FUNCTION_BLOCK "SimaHydTO_AxisAdvanced_SyncAxis"   // FB33112, FBD
TITLE = SimaHydTO_AxisAdvanced_SyncAxis
{ S7_Optimized_Access := 'TRUE' }
FAMILY : SimaHydTO/LAxisBasics
VERSION : 1.0
// Function block information: See Function block network 1
// stored: AutoNumber true, IsIECCheckEnabled false, IsRetainMemResEnabled false, MemoryReserve 100, SetENOAutomatically false, UDAEnableTagReadback false
   VAR_INPUT
      axis : TO_SynchronousAxis;   // Technology object (axis)
      moveRelativeExecute : Bool;   // MC_MoveRelative: Start job with a positive edge
      moveRelativeDistance : LReal := 0.0;   // Distance of relative movement
      moveAbsoluteExecute : Bool;   // MC_MoveAbsolute: Start job with a positive edge
      moveAbsolutePosition : LReal := 0.0;   // Target position of absolute movement
      moveAbsoluteDirection : Int := 1;   // Direction of absolute movement: 0: Positive direction / 1: Negative direction / 3: Shortest direction
      moveAbsPositionControlled : Bool := true;   // 0: Non position-controlled operation / 1: Position-controlled mode - The parameter applies as long as the MC_MoveJog command is executed. After this, the setting of MC_Power applies again.
      haltExecute : Bool;   // MC_Halt: Start job with a positive edge
      haltAbortAcceleration : Bool := false;   // Acceleration control: False: The current acceleration at the start of the job is reduced using the configured jerk. Afterwards, the deceleration builds up / True: The acceleration is set to 0.0 at the start of the job, and the deceleration immediately builds up.
      Velocity : LReal := 100.0;   // Velocity of movement
      Acceleration : LReal := -1.0;   // Acceleration of movement
      Deceleration : LReal := -1.0;   // Deceleration of movement
      Jerk : LReal := -1.0;   // Jerk of movement
   END_VAR
   VAR_OUTPUT
      moveRelativeDone { ExternalWritable := 'False'} : Bool;   // MC_MoveRelative: Job is completed
      moveRelativeBusy { ExternalWritable := 'False'} : Bool;   // MC_MoveRelative: Job is running
      moveAbsoluteDone { ExternalWritable := 'False'} : Bool;   // MC_MoveAbsolute: Job is completed
      moveAbsoluteBusy { ExternalWritable := 'False'} : Bool;   // MC_MoveAbsolute: Job is running
      haltDone { ExternalWritable := 'False'} : Bool;   // MC_Halt: Job is running
      haltBusy { ExternalWritable := 'False'} : Bool;   // MC_Halt: Job is running
      commandAborted { ExternalWritable := 'False'} : Bool;   // The job was aborted by another job during execution (see also StatusID)
      error { ExternalWritable := 'False'} : Bool;   // An error occurred during execution of the job. The job is rejected. The cause of the error can be found in the "ErrorID" parameter.
      errorID { ExternalWritable := 'False'} : Word;   // ErrorID of motion control instruction (see also StatusID)
      statusID { ExternalWritable := 'False'} : Int;   // Additional specification of affected Motion control instruction of CommandAborted or Error: 0: No instruction / 1: MC_Power / 2: MC_Reset / 3: MC_Home / 4: MC_MoveJog
   END_VAR
   VAR
      instMcMoveRelative { ExternalAccessible := 'False'; ExternalVisible := 'False'; ExternalWritable := 'False'; S7_SetPoint := 'True'} : MC_MOVERELATIVE;   // PLCopen functions of basic motion control
      instMcMoveAbsolute { ExternalAccessible := 'False'; ExternalVisible := 'False'; ExternalWritable := 'False'; S7_SetPoint := 'True'} : MC_MOVEABSOLUTE;
      instMcHalt { ExternalAccessible := 'False'; ExternalVisible := 'False'; ExternalWritable := 'False'; S7_SetPoint := 'True'} : MC_HALT;
      statCommandAborted { ExternalAccessible := 'False'; ExternalVisible := 'False'; ExternalWritable := 'False'} : Array[#ARRAY_BEGIN..#ARRAY_END] of Bool;   // Arrays to save error information of PLCopen functions
      statError { ExternalAccessible := 'False'; ExternalVisible := 'False'; ExternalWritable := 'False'} : Array[#ARRAY_BEGIN..#ARRAY_END] of Bool;
      statErrorID { ExternalAccessible := 'False'; ExternalVisible := 'False'; ExternalWritable := 'False'} : Array[#ARRAY_BEGIN..#ARRAY_END] of Word;
      instMoveAbsOpenLoop { ExternalAccessible := 'False'; ExternalVisible := 'False'; ExternalWritable := 'False'; S7_SetPoint := 'True'} : "LSimaHydTO_MC_MoveAbsOpenLoop";
   END_VAR
   VAR_TEMP
      tempDwordCommandAborted : DWord;   // Variables to check error informations of PLCopen functions
      tempDwordError : DWord;
      tempCount : Int;   // Counter of FOR counting loop
   END_VAR
   VAR CONSTANT
      ARRAY_BEGIN : Int := 1;   // Start-Index of array (Maximum 32 Array elements!)
      ARRAY_END : Int := 32;   // End-Index of array (Maximum 32 Array elements!)
      ERROR_DEFAULT : Bool := false;   // Default values of output signals
      ERRORID_DEFAULT : Word := 16#0;
      STATUSID_DEFAULT : Int := 0;
   END_VAR
BEGIN

REGION Network 1 (SCL): Axis Basics - Header
   //=============================================================================
   //SIEMENS AG
   //(c)Copyright 2016 All Rights Reserved
   //-----------------------------------------------------------------------------
   //Library:       AxisAdvanced
   //Tested with:   S7-1500 V2.5
   //Engineering:   TIA Portal V15
   //Restrictions:  Motion Control Library V4.0
   //Requirements:  S7-1500(T)
   //Functionality: Advanced axis control of TO_SynchronousAxis
   //-----------------------------------------------------------------------------
   //Change log table:
   //Version  Date       Expert in charge Changes applied
   //01.00.00 19.07.2019 ArSc             First released version
   //=============================================================================
END_REGION

REGION Network 2: Axis Advanced - MC_MoveRelative
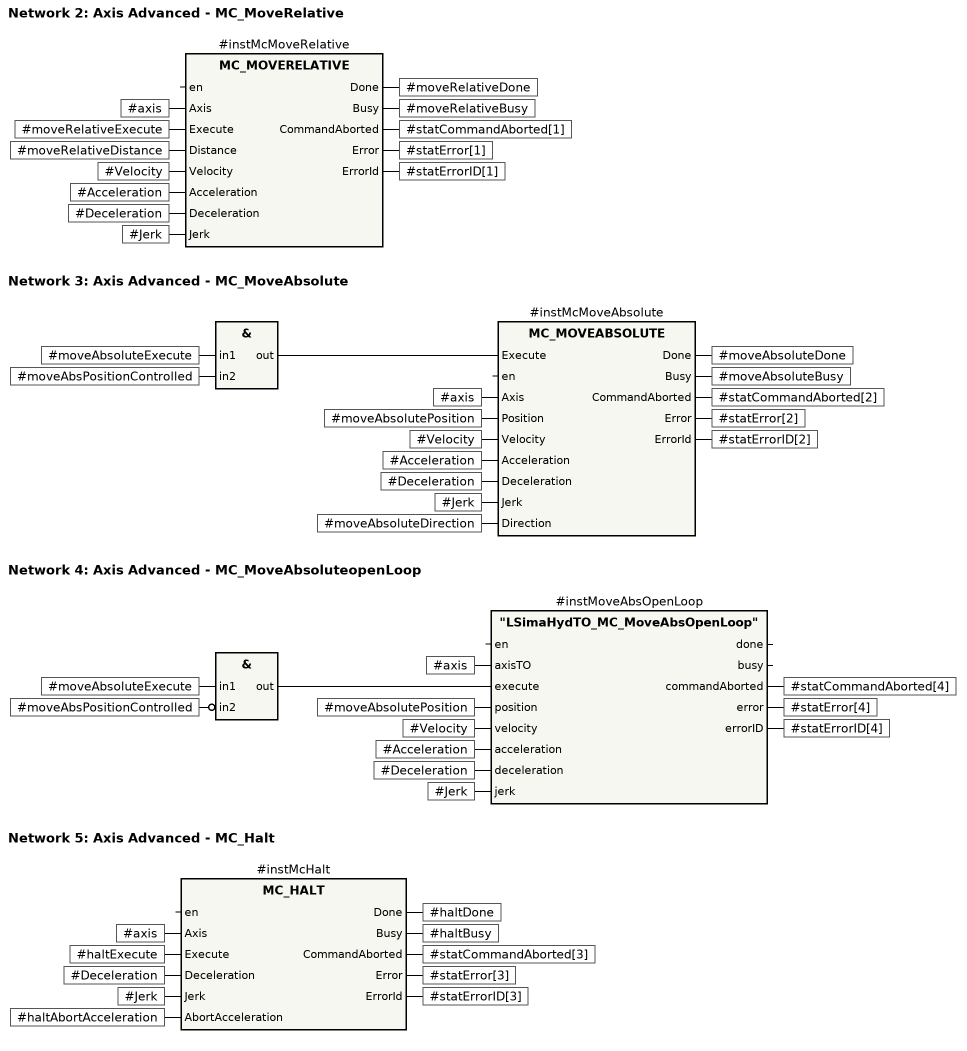
   #instMcMoveRelative(Axis := #axis,   // MC_MOVERELATIVE
                       Execute := #moveRelativeExecute,
                       Distance := #moveRelativeDistance,
                       Velocity := #Velocity,
                       Acceleration := #Acceleration,
                       Deceleration := #Deceleration,
                       Jerk := #Jerk,
                       Done => #moveRelativeDone,
                       Busy => #moveRelativeBusy,
                       CommandAborted => #statCommandAborted[1],
                       Error => #statError[1],
                       ErrorId => #statErrorID[1]);
END_REGION

REGION Network 3: Axis Advanced - MC_MoveAbsolute
   #instMcMoveAbsolute(Execute := #moveAbsoluteExecute AND #moveAbsPositionControlled,   // MC_MOVEABSOLUTE
                       Axis := #axis,
                       Position := #moveAbsolutePosition,
                       Velocity := #Velocity,
                       Acceleration := #Acceleration,
                       Deceleration := #Deceleration,
                       Jerk := #Jerk,
                       Direction := #moveAbsoluteDirection,
                       Done => #moveAbsoluteDone,
                       Busy => #moveAbsoluteBusy,
                       CommandAborted => #statCommandAborted[2],
                       Error => #statError[2],
                       ErrorId => #statErrorID[2]);
END_REGION

REGION Network 4: Axis Advanced - MC_MoveAbsoluteopenLoop
   #instMoveAbsOpenLoop(axisTO := #axis,   // "LSimaHydTO_MC_MoveAbsOpenLoop"
                        execute := #moveAbsoluteExecute AND NOT #moveAbsPositionControlled,
                        position := #moveAbsolutePosition,
                        velocity := #Velocity,
                        acceleration := #Acceleration,
                        deceleration := #Deceleration,
                        jerk := #Jerk,
                        commandAborted => #statCommandAborted[4],
                        error => #statError[4],
                        errorID => #statErrorID[4]);
END_REGION

REGION Network 5: Axis Advanced - MC_Halt
   #instMcHalt(Axis := #axis,   // MC_HALT
               Execute := #haltExecute,
               Deceleration := #Deceleration,
               Jerk := #Jerk,
               AbortAcceleration := #haltAbortAcceleration,
               Done => #haltDone,
               Busy => #haltBusy,
               CommandAborted => #statCommandAborted[3],
               Error => #statError[3],
               ErrorId => #statErrorID[3]);
END_REGION

REGION Network 6 (SCL): Axis Basics - Generate output signals and error detection
   //General output signals

   //Reset output signals
   #commandAborted := False;
   #error := False;
   #errorID := #ERRORID_DEFAULT;
   #statusID := #STATUSID_DEFAULT;

   //Transfer ARRAY to DWORD
   GATHER(IN:=#statCommandAborted,
          OUT=>#tempDwordCommandAborted);
   GATHER(IN:=#statError,
          OUT=>#tempDwordError);

   //Check for errors or command aborts
   IF (#tempDwordError > DWORD#0)
   THEN
     //Select error information
     FOR #tempCount := #ARRAY_BEGIN TO #ARRAY_END
     DO
       IF (#statError[#tempCount] = True)
       THEN
         #error := True;
         #errorID := #statErrorID[#tempCount];
         #statusID := #tempCount;
         EXIT;
       END_IF;
     END_FOR;
   ELSIF (#tempDwordCommandAborted > DWORD#0)
   THEN
     //Select command aborted information
     FOR #tempCount := #ARRAY_BEGIN TO #ARRAY_END
     DO
       IF (#statCommandAborted[#tempCount] = True)
       THEN
         #commandAborted := True;
         #errorID := #statErrorID[#tempCount];
         #statusID := #tempCount;
         EXIT;
       END_IF;
     END_FOR;
   END_IF;
END_REGION
END_FUNCTION_BLOCK

FUNCTION_BLOCK "SimaHydTO_ParameterSettings"
{ S7_Optimized_Access := 'TRUE' }
FAMILY : SimaHydTO
VERSION : 1.0
   VAR_IN_OUT 
      hmiConnection : "SimaHydTO_typeHMIConnection";
      axisData : "LSimaHydTO_typeAxisData";
      VCharArray : Array[*] of "SimaHydTO_typeVCharArray";
   END_VAR

   VAR 
      statSaveDBL { ExternalAccessible := 'False'; ExternalVisible := 'False'; ExternalWritable := 'False'} : Bool;
      statLoadDBL { ExternalAccessible := 'False'; ExternalVisible := 'False'; ExternalWritable := 'False'} : Bool;
      statEditOld { ExternalAccessible := 'False'; ExternalVisible := 'False'; ExternalWritable := 'False'} : Bool;
      statActivateOld { ExternalAccessible := 'False'; ExternalVisible := 'False'; ExternalWritable := 'False'} : Bool;
      statAbortOld { ExternalAccessible := 'False'; ExternalVisible := 'False'; ExternalWritable := 'False'} : Bool;
      statRestoreOld { ExternalAccessible := 'False'; ExternalVisible := 'False'; ExternalWritable := 'False'} : Bool;
      statApplayOld { ExternalAccessible := 'False'; ExternalVisible := 'False'; ExternalWritable := 'False'} : Bool;
      statDefaultAxisData { ExternalAccessible := 'False'; ExternalVisible := 'False'; ExternalWritable := 'False'} : "SimaHydTO_typeHMIConnectionParameterSettingsAxisData";
      instMC_WriteToROM { ExternalAccessible := 'False'; ExternalVisible := 'False'; ExternalWritable := 'False'} : "LSimaHydTO_MC_WriteToROM";
      instMC_ReadFromROM { ExternalAccessible := 'False'; ExternalVisible := 'False'; ExternalWritable := 'False'} : "LSimaHydTO_MC_ReadFromROM";
      instVCharSelector { ExternalAccessible := 'False'; ExternalVisible := 'False'; ExternalWritable := 'False'} : "SimaHydTO_HmiVCharSelector";
      statSaveOld { ExternalAccessible := 'False'; ExternalVisible := 'False'; ExternalWritable := 'False'} : Bool;
   END_VAR

   VAR_TEMP 
      tempVariant : Variant;
      tempErrorVariant : Int;
      tempDbAny : DB_ANY;
      tempVCharData : REF_TO "LSimaHydTO_typeVCharData";
   END_VAR


BEGIN
	//=============================================================================
	//SIEMENS AG
	//(c)Copyright 2016 All Rights Reserved
	//-----------------------------------------------------------------------------
	//Library:       SimaHydTO_ParameterSettings
	//Tested with:   S7-1500 V2.5
	//Engineering:   TIA Portal V15
	//Restrictions:  -
	//Requirements:  S7-1500(T)
	//Functionality: Manipulate parameter data of selected hydraulic axis
	//-----------------------------------------------------------------------------
	//Change log table:
	//Version  Date       Expert in charge Changes applied
	//01.00.00 17.07.2019 ArSc             First released version
	//=============================================================================
	
	
	IF (#hmiConnection.AxisSelector.Status.selectionChanged
	    OR #instMC_ReadFromROM.done)
	    OR (#hmiConnection.ParameterSettings.Commands.Edit
	    AND NOT #statEditOld
	    AND NOT #hmiConnection.ParameterSettings.Status.EditorActive)
	THEN
	    IF #hmiConnection.AxisSelector.Status.dataValid THEN
	        //Convert data
	        //Get data from axis
	        #hmiConnection.ParameterSettings.AxisData.Actor := #axisData.Actor;
	        #hmiConnection.ParameterSettings.AxisData.ValveCharacteristic := #axisData.ValveCharacteristic;
	        #hmiConnection.ParameterSettings.AxisData.ForceLimits := #axisData.ForceLimits;
	        #hmiConnection.ParameterSettings.AxisData.Pressure_A_Transducer := #axisData.Pressure_A_Transducer;
	        #hmiConnection.ParameterSettings.AxisData.Pressure_B_Transducer := #axisData.Pressure_B_Transducer;
	        #hmiConnection.ParameterSettings.AxisData.PositionControl := #axisData.PositionControl;
	        #hmiConnection.ParameterSettings.AxisData.ForceControl := #axisData.ForceControl;
	        #hmiConnection.ParameterSettings.AxisData.DynamicAxisModel := #axisData.DynamicAxisModel;
	        #hmiConnection.ParameterSettings.AxisData.SmoothingFilter := #axisData.SmoothingFilter;
	        #hmiConnection.ParameterSettings.AxisData.Name := #axisData.Name;
	        IF #axisData.ValveCharacteristic.DB_NUMBER > 0 THEN
	            #tempDbAny := #axisData.ValveCharacteristic.DB_NUMBER;
	            #tempVariant := DB_ANY_TO_VARIANT(in := #tempDbAny, err => #tempErrorVariant);
	            
	            IF TypeOf(#tempVariant) = LSimaHydTO_typeVCharData THEN
	                #tempVCharData ?= #tempVariant;
	                #hmiConnection.ParameterSettings.AxisData.VCharName := #tempVCharData^.Name;
	            ELSE
	                #hmiConnection.ParameterSettings.AxisData.VCharName := wstring#'';
	            END_IF;
	        ELSE
	            #hmiConnection.ParameterSettings.AxisData.VCharName := wstring#'';
	        END_IF;
	        
	    ELSE
	        #hmiConnection.ParameterSettings.AxisData := #statDefaultAxisData;
	    END_IF;
	    IF #hmiConnection.AxisSelector.Status.selectionChanged THEN
	        #hmiConnection.ParameterSettings.Status.EditorActive := False;
	    END_IF;
	    
	END_IF;
	
	//Open parameter data
	IF (#hmiConnection.ParameterSettings.Commands.Edit
	    AND NOT #statEditOld
	    AND NOT #hmiConnection.ParameterSettings.Status.EditorActive
	    AND #hmiConnection.AxisSelector.Status.dataValid)
	THEN
	    #hmiConnection.ParameterSettings.Status.EditorActive := True;
	END_IF;
	
	//Save parameter data
	IF ((#hmiConnection.ParameterSettings.Commands.Activate AND NOT #statActivateOld)
	    OR (#hmiConnection.ParameterSettings.Commands.Save AND NOT #statSaveOld))
	    AND #hmiConnection.ParameterSettings.Status.EditorActive
	    AND #hmiConnection.AxisSelector.Status.dataValid
	THEN
	    //Write back axis data
	    #hmiConnection.ParameterSettings.Status.StateActivation := 1;
	    
	    #axisData.Actor := #hmiConnection.ParameterSettings.AxisData.Actor;
	    #axisData.ValveCharacteristic := #hmiConnection.ParameterSettings.AxisData.ValveCharacteristic;
	    #axisData.ForceLimits := #hmiConnection.ParameterSettings.AxisData.ForceLimits;
	    #axisData.Pressure_A_Transducer := #hmiConnection.ParameterSettings.AxisData.Pressure_A_Transducer;
	    #axisData.Pressure_B_Transducer := #hmiConnection.ParameterSettings.AxisData.Pressure_B_Transducer;
	    #axisData.PositionControl := #hmiConnection.ParameterSettings.AxisData.PositionControl;
	    #axisData.ForceControl := #hmiConnection.ParameterSettings.AxisData.ForceControl;
	    #axisData.DynamicAxisModel := #hmiConnection.ParameterSettings.AxisData.DynamicAxisModel;
	    #axisData.SmoothingFilter := #hmiConnection.ParameterSettings.AxisData.SmoothingFilter;
	    #axisData.Name := #hmiConnection.ParameterSettings.AxisData.Name;
	    //  save to load memory
	    #hmiConnection.ParameterSettings.Status.EditorActive := False;
	    #hmiConnection.ParameterSettings.Status.StateActivation := 0;
	    #hmiConnection.ParameterSettings.Status.StateLoading := 0;
	END_IF;
	
	IF #hmiConnection.ParameterSettings.Commands.Save
	    //AND #hmiConnection.ParameterSettings.Status.StateActivation = 1
	    AND #hmiConnection.AxisSelector.Status.dataValid
	    AND NOT #statSaveOld
	THEN
	    #statSaveDBL := TRUE;
	    
	END_IF;
	
	#instMC_WriteToROM(execute := #statSaveDBL,
	                   axis := #axisData);
	
	IF #instMC_WriteToROM.busy THEN
	    #hmiConnection.ParameterSettings.Status.StateSaving := 1;
	ELSIF #instMC_WriteToROM.error THEN
	    #hmiConnection.ParameterSettings.Status.StateSaving := 2;
	    #statSaveDBL := FALSE;
	    
	ELSE
	    #hmiConnection.ParameterSettings.Status.StateSaving := 0;
	    #statSaveDBL := FALSE;
	    
	END_IF;
	
	
	IF (#hmiConnection.ParameterSettings.Commands.Restore
	    AND NOT #statRestoreOld)
	    AND #hmiConnection.AxisSelector.Status.dataValid
	THEN
	    #hmiConnection.ParameterSettings.Status.StateActivation := 0;
	    #hmiConnection.ParameterSettings.Status.StateSaving := 0;
	    #hmiConnection.ParameterSettings.Status.StateLoading := 1;
	    
	    #statLoadDBL := true;
	END_IF;
	#instMC_ReadFromROM(execute := #statLoadDBL,
	                    axis := #axisData);
	
	IF NOT #instMC_ReadFromROM.busy THEN
	    IF #instMC_ReadFromROM.done THEN
	        #hmiConnection.ParameterSettings.Status.StateActivation := 0;
	        #hmiConnection.ParameterSettings.Status.StateLoading := 0;
	    ELSIF #instMC_ReadFromROM.error THEN
	        #hmiConnection.ParameterSettings.Status.StateLoading := 2;
	    END_IF;
	    
	    
	    #statLoadDBL := FALSE;
	END_IF;
	
	
	//Abort parameter data
	IF (#hmiConnection.ParameterSettings.Commands.Abort
	    AND #hmiConnection.ParameterSettings.Status.EditorActive)
	THEN
	    //Reset output singal
	    #hmiConnection.ParameterSettings.Status.EditorActive := False;
	END_IF;
	
	
	//Save data from last cycle
	#statAbortOld := #hmiConnection.ParameterSettings.Commands.Abort;
	#statActivateOld := #hmiConnection.ParameterSettings.Commands.Activate;
	#statEditOld := #hmiConnection.ParameterSettings.Commands.Edit;
	#statRestoreOld := #hmiConnection.ParameterSettings.Commands.Restore;
	#statSaveOld := #hmiConnection.ParameterSettings.Commands.Save;
	
END_FUNCTION_BLOCK

FUNCTION_BLOCK "LSimaHydTO_MC_WriteToROM"
{ S7_Optimized_Access := 'TRUE' }
AUTHOR : APC_ERLF
FAMILY : LSimaHydTO
VERSION : 1.0
   VAR_INPUT 
      execute : Bool;
      parameter : Int;
   END_VAR

   VAR_OUTPUT 
      busy { ExternalWritable := 'False'} : Bool;
      done { ExternalWritable := 'False'} : Bool;
      commandAborted { ExternalWritable := 'False'} : Bool;
      error { ExternalWritable := 'False'} : Bool;
      errorID { ExternalWritable := 'False'} : Int;
   END_VAR

   VAR_IN_OUT 
      axis : "LSimaHydTO_typeAxisData";
   END_VAR

   VAR 
      statState { ExternalAccessible := 'False'; ExternalVisible := 'False'; ExternalWritable := 'False'} : DInt;
      statExecuteOld { ExternalAccessible := 'False'; ExternalVisible := 'False'; ExternalWritable := 'False'} : Bool;
      statBusyWrit { ExternalAccessible := 'False'; ExternalVisible := 'False'; ExternalWritable := 'False'} : Bool;
      statBusy { ExternalAccessible := 'False'; ExternalVisible := 'False'; ExternalWritable := 'False'} : Bool;
      statRetVal { ExternalAccessible := 'False'; ExternalVisible := 'False'; ExternalWritable := 'False'} : Int;
   END_VAR

   VAR_TEMP 
      tempVarParameter : Variant;
   END_VAR

   VAR CONSTANT 
      STATE_IDLE : DInt := 0;
      LAST_PARAM : DInt := 10;
   END_VAR


BEGIN
	//================================================================================
	//SIEMENS AG // (c)Copyright 2019 All Rights Reserved
	//--------------------------------------------------------------------------------
	//Library:       LSimaHydTO
	//Tested with:   S7-15xx
	//Engineering:   TIA Portal  V15
	//Restrictions:  -
	//Requirements:  S7-1500 (FW 2.5)
	//Functionality: Write parameter from RAM into ROM 
	//
	//--------------------------------------------------------------------------------
	//Change log table:
	//
	//Version     Date          Expert in charge    Changes applied
	//01.00.00    15.03.2018    APC_ERLF            First released version
	//================================================================================
	
	
	IF #execute AND NOT #statExecuteOld THEN
	  #done := FALSE;
	  #statBusy := TRUE;
	  #statBusyWrit := FALSE;
	  #error := FALSE;
	  #errorID := 0;
	  IF #parameter = 0 OR #parameter = 1 THEN
	    #statState := 1;
	  ELSE
	    #statState := #parameter;
	  END_IF;
	END_IF;
	IF #statBusy THEN
	  
	  CASE #statState OF
	      
	    1: // actor
	      
	      #statRetVal := WRIT_DBL(REQ := TRUE, SRCBLK := #axis.Actor, BUSY => #statBusyWrit, DSTBLK => #axis.Actor);
	      
	      
	    2: // valve characteristic
	      
	      #statRetVal := WRIT_DBL(REQ := TRUE, SRCBLK := #axis.ValveCharacteristic, BUSY => #statBusyWrit, DSTBLK => #axis.ValveCharacteristic);
	      
	      
	    3: // force limits
	      
	      #statRetVal := WRIT_DBL(REQ := TRUE, SRCBLK := #axis.ForceLimits, BUSY => #statBusyWrit, DSTBLK => #axis.ForceLimits);
	      
	      
	    4: // A-transducer
	      
	      #statRetVal := WRIT_DBL(REQ := TRUE, SRCBLK := #axis.Pressure_A_Transducer, BUSY => #statBusyWrit, DSTBLK => #axis.Pressure_A_Transducer);
	      
	      
	    5: // B-transducer
	      
	      #statRetVal := WRIT_DBL(REQ := TRUE, SRCBLK := #axis.Pressure_B_Transducer, BUSY => #statBusyWrit, DSTBLK => #axis.Pressure_B_Transducer);
	      
	      
	    6: // position control
	      
	      #statRetVal := WRIT_DBL(REQ := TRUE, SRCBLK := #axis.PositionControl, BUSY => #statBusyWrit, DSTBLK => #axis.PositionControl);
	      
	      
	    7: // force control
	      
	      #statRetVal := WRIT_DBL(REQ := TRUE, SRCBLK := #axis.ForceControl, BUSY => #statBusyWrit, DSTBLK => #axis.ForceControl);
	      
	      
	    8: // dynamic axis model
	      
	      #statRetVal := WRIT_DBL(REQ := TRUE, SRCBLK := #axis.DynamicAxisModel, BUSY => #statBusyWrit, DSTBLK => #axis.DynamicAxisModel);
	      
	      
	    9: // smoothing filter
	      
	      #statRetVal := WRIT_DBL(REQ := TRUE, SRCBLK := #axis.SmoothingFilter, BUSY => #statBusyWrit, DSTBLK => #axis.SmoothingFilter);
	      
	      
	    10: // name
	      
	      #statRetVal := WRIT_DBL(REQ := TRUE, SRCBLK := #axis.Name, BUSY => #statBusyWrit, DSTBLK => #axis.Name);
	      
	      
	    ELSE
	      #statState := #STATE_IDLE;
	      #statBusy := FALSE;
	  END_CASE;
	  
	  IF NOT #statBusyWrit THEN
	    IF #statRetVal = 0 THEN
	      IF #parameter = 0 AND #statState < #LAST_PARAM THEN
	        #statState := 1 + #statState;
	      ELSE
	        #statBusy := false;
	        #done := TRUE;
	      END_IF;
	    ELSE
	      #statBusy := FALSE;
	      #error := TRUE;
	      #errorID := #statRetVal;
	      #statState := #STATE_IDLE;
	    END_IF;
	  END_IF;
	ELSIF NOT #execute THEN
	  #done := FALSE;
	  #error := FALSE;
	  #errorID := 0;
	END_IF;
	#statExecuteOld := #execute;
	#busy := #statBusy;
	
END_FUNCTION_BLOCK

FUNCTION_BLOCK "LSimaHydTO_MC_ReadFromROM"
{ S7_Optimized_Access := 'TRUE' }
AUTHOR : APC_ERLF
FAMILY : LSimaHydTO
VERSION : 1.0
   VAR_INPUT 
      execute : Bool;
      parameter : Int;
   END_VAR

   VAR_OUTPUT 
      busy { ExternalWritable := 'False'} : Bool;
      done { ExternalWritable := 'False'} : Bool;
      commandAborted { ExternalWritable := 'False'} : Bool;
      error { ExternalWritable := 'False'} : Bool;
      errorID { ExternalWritable := 'False'} : Word;
   END_VAR

   VAR_IN_OUT 
      axis : "LSimaHydTO_typeAxisData";
   END_VAR

   VAR 
      statState { ExternalAccessible := 'False'; ExternalVisible := 'False'; ExternalWritable := 'False'} : DInt;
      statExecuteOld { ExternalAccessible := 'False'; ExternalVisible := 'False'; ExternalWritable := 'False'} : Bool;
      statBusyRead { ExternalAccessible := 'False'; ExternalVisible := 'False'; ExternalWritable := 'False'} : Bool;
      statRetVal { ExternalAccessible := 'False'; ExternalVisible := 'False'; ExternalWritable := 'False'} : Int;
   END_VAR

   VAR_TEMP 
      tempVarParameter : Variant;
   END_VAR

   VAR CONSTANT 
      STATE_IDLE : DInt := 0;
      LAST_PARAM : DInt := 10;
   END_VAR


BEGIN
	//================================================================================
	//SIEMENS AG // (c)Copyright 2019 All Rights Reserved
	//--------------------------------------------------------------------------------
	//Library:       LSimaHydTO
	//Tested with:   S7-15xx
	//Engineering:   TIA Portal  V15
	//Restrictions:  -
	//Requirements:  S7-1500 (FW 2.5)
	//Functionality: Read parameter from ROM into RAM 
	//
	//--------------------------------------------------------------------------------
	//Change log table:
	//
	//Version     Date          Expert in charge    Changes applied
	//01.00.00    15.03.2018    APC_ERLF            First released version
	//================================================================================
	
	
	IF #execute AND NOT #statExecuteOld THEN
	  #done := FALSE;
	  #busy := TRUE;
	  #statBusyRead := TRUE;
	  #error := FALSE;
	  #errorID := 0;
	  IF #parameter = 0 OR #parameter = 1 THEN
	    #statState := 1;
	  ELSE
	    #statState := #parameter;
	  END_IF;
	END_IF;
	IF #statBusyRead THEN
	  
	  CASE #statState OF
	      
	    1: // actor
	      
	      #statRetVal := READ_DBL(REQ := TRUE, SRCBLK := #axis.Actor, BUSY => #statBusyRead, DSTBLK => #axis.Actor);
	      
	      
	    2: // valve characteristic
	      
	      #statRetVal := READ_DBL(REQ := TRUE, SRCBLK := #axis.ValveCharacteristic, BUSY => #statBusyRead, DSTBLK => #axis.ValveCharacteristic);
	      
	      
	    3: // force limits
	      
	      #statRetVal := READ_DBL(REQ := TRUE, SRCBLK := #axis.ForceLimits, BUSY => #statBusyRead, DSTBLK => #axis.ForceLimits);
	      
	      
	    4: // ring transducer
	      
	      #statRetVal := READ_DBL(REQ := TRUE, SRCBLK := #axis.Pressure_A_Transducer, BUSY => #statBusyRead, DSTBLK => #axis.Pressure_A_Transducer);
	      
	      
	    5: // piston transducer
	      
	      #statRetVal := READ_DBL(REQ := TRUE, SRCBLK := #axis.Pressure_B_Transducer, BUSY => #statBusyRead, DSTBLK => #axis.Pressure_B_Transducer);
	      
	      
	    6: // position control
	      
	      #statRetVal := READ_DBL(REQ := TRUE, SRCBLK := #axis.PositionControl, BUSY => #statBusyRead, DSTBLK => #axis.PositionControl);
	      
	      
	    7: // force control
	      
	      #statRetVal := READ_DBL(REQ := TRUE, SRCBLK := #axis.ForceControl, BUSY => #statBusyRead, DSTBLK => #axis.ForceControl);
	      
	      
	    8: // dynamic axis model
	      
	      #statRetVal := READ_DBL(REQ := TRUE, SRCBLK := #axis.DynamicAxisModel, BUSY => #statBusyRead, DSTBLK => #axis.DynamicAxisModel);
	      
	      
	    9: // smoothing filter
	      
	      #statRetVal := READ_DBL(REQ := TRUE, SRCBLK := #axis.SmoothingFilter, BUSY => #statBusyRead, DSTBLK => #axis.SmoothingFilter);
	      
	      
	    10: // name
	      
	      #statRetVal := READ_DBL(REQ := TRUE, SRCBLK := #axis.Name, BUSY => #statBusyRead, DSTBLK => #axis.Name);
	      
	      
	    ELSE
	      #statState := #STATE_IDLE;
	      #statBusyRead := FALSE;
	  END_CASE;
	  
	  IF NOT #statBusyRead THEN
	    IF #statRetVal = 0 THEN
	      IF #parameter = 0 AND #statState < #LAST_PARAM THEN
	        #statState := 1 + #statState;
	        #statBusyRead := TRUE;
	      ELSE
	        #busy := false;
	        #done := TRUE;
	      END_IF;
	    ELSE
	      #busy := FALSE;
	      #error := TRUE;
	      #errorID := INT_TO_WORD(#statRetVal);
	      #statState := #STATE_IDLE;
	    END_IF;
	  END_IF;
	ELSIF NOT #execute THEN
	  #done := FALSE;
	  #error := FALSE;
	  #errorID := 0;
	END_IF;
	#statExecuteOld := #execute;
	
END_FUNCTION_BLOCK

FUNCTION_BLOCK "SimaHydTO_FindObjects"
{ S7_Optimized_Access := 'TRUE' }
FAMILY : SimaHydTO
VERSION : 1.0
   VAR_INPUT 
      execute : Bool;
   END_VAR

   VAR_OUTPUT 
      done { ExternalWritable := 'False'} : Bool;
      busy { ExternalWritable := 'False'} : Bool;
      error { ExternalWritable := 'False'} : Bool;
      status { ExternalWritable := 'False'} : Word := #STATUS_NO_CALL;
   END_VAR

   VAR_IN_OUT 
      axesArray : Array[*] of "SimaHydTO_typeAxesArray";
      vCharArray : Array[*] of "SimaHydTO_typeVCharArray";
   END_VAR

   VAR 
      statAxesArrMinIndex { ExternalAccessible := 'False'; ExternalVisible := 'False'; ExternalWritable := 'False'} : Int;
      statAxesArrMaxIndex { ExternalAccessible := 'False'; ExternalVisible := 'False'; ExternalWritable := 'False'} : Int;
      statVCharArrMinIndex { ExternalAccessible := 'False'; ExternalVisible := 'False'; ExternalWritable := 'False'} : Int;
      statVCharArrMaxIndex { ExternalAccessible := 'False'; ExternalVisible := 'False'; ExternalWritable := 'False'} : Int;
      statVCharArrayFull { ExternalAccessible := 'False'; ExternalVisible := 'False'; ExternalWritable := 'False'} : Bool;
      statAxesArrayFull { ExternalAccessible := 'False'; ExternalVisible := 'False'; ExternalWritable := 'False'} : Bool;
      statExecuteOld { ExternalAccessible := 'False'; ExternalVisible := 'False'; ExternalWritable := 'False'} : Bool;
      statDone { ExternalAccessible := 'False'; ExternalVisible := 'False'; ExternalWritable := 'False'} : Bool;
      statBusy { ExternalAccessible := 'False'; ExternalVisible := 'False'; ExternalWritable := 'False'} : Bool;
      statError { ExternalAccessible := 'False'; ExternalVisible := 'False'; ExternalWritable := 'False'} : Bool;
      statStatus { ExternalAccessible := 'False'; ExternalVisible := 'False'; ExternalWritable := 'False'} : Word := #STATUS_NO_CALL;
      statFBState { ExternalAccessible := 'False'; ExternalVisible := 'False'; ExternalWritable := 'False'} : DInt := #FB_STATE_NO_PROCESSING;
      statActDB_NUMBER { ExternalAccessible := 'False'; ExternalVisible := 'False'; ExternalWritable := 'False'} : UInt;
      statRunTime { ExternalAccessible := 'False'; ExternalVisible := 'False'; ExternalWritable := 'False'} : LReal;
      statMemStart { ExternalAccessible := 'False'; ExternalVisible := 'False'; ExternalWritable := 'False'} : LReal;
      statMem { ExternalAccessible := 'False'; ExternalVisible := 'False'; ExternalWritable := 'False'} : LReal;
   END_VAR

   VAR_TEMP 
      tempExecute : Bool;
      tempInt : Int;
      tempInitDone : Bool;
   END_VAR

   VAR CONSTANT 
      FB_STATE_NO_PROCESSING : DInt := 0;
      FB_STATE_PROCESSING : DInt := 2;
      STATUS_EXECUTION_FINISHED : Word := 16#0000;
      STATUS_NO_CALL : Word := 16#7000;
      STATUS_FIRST_CALL : Word := 16#7001;
      STATUS_SUBSEQUENT_CALL : Word := 16#7002;
      ERR_UNDEFINED_STATE : Word := 16#8600;
   END_VAR


BEGIN
	//=============================================================================
	//SIEMENS AG
	//(c)Copyright 2016 All Rights Reserved
	//-----------------------------------------------------------------------------
	//Library:       SimaHydTO_HMI
	//Tested with:   S7-1500 V2.5
	//Engineering:   TIA Portal V15
	//Restrictions:  -
	//Requirements:  S7-1500(T)
	//Functionality: Search for hydraulic axes and valve charachteristics in project
	//-----------------------------------------------------------------------------
	//Change log table:
	//Version  Date       Expert in charge Changes applied
	//01.00.00 12.07.2019 ArSc             First released version
	//=============================================================================
	
	#tempExecute := #execute; // Work with temporary value / create process image
	
	REGION TRIGGERING
	    IF (#tempExecute = TRUE) AND (#statExecuteOld = FALSE) // Check if FB is triggered
	        
	    THEN // First call; initialize FB
	        #statDone := FALSE;
	        #statBusy := TRUE;
	        #statError := FALSE;
	        #statStatus := #STATUS_FIRST_CALL;
	        
	        #statAxesArrMinIndex := DINT_TO_INT(LOWER_BOUND(ARR := #axesArray, DIM := 1));
	        #statAxesArrMaxIndex := DINT_TO_INT(UPPER_BOUND(ARR := #axesArray, DIM := 1));
	        #statVCharArrMinIndex := DINT_TO_INT(LOWER_BOUND(ARR := #vCharArray, DIM := 1));
	        #statVCharArrMaxIndex := DINT_TO_INT(UPPER_BOUND(ARR := #vCharArray, DIM := 1));
	        
	        #statVCharArrayFull := FALSE;
	        #statAxesArrayFull := FALSE;
	        #statActDB_NUMBER := 1;
	        
	        #statFBState := #FB_STATE_PROCESSING; // State machine - start processing
	        
	    ELSIF (#statStatus = #STATUS_FIRST_CALL) THEN
	        #statStatus := #STATUS_SUBSEQUENT_CALL;
	    END_IF;
	    
	    // Edge detection 'execute' input
	    #statExecuteOld := #tempExecute;
	END_REGION TRIGGERING
	
	IF (#statStatus = #STATUS_NO_CALL) THEN // Nothing to do -> End here to reduce "system load"
	    RETURN;
	END_IF;
	
	REGION STATE_MACHINE
	    CASE #statFBState OF // State machine of FB
	        #FB_STATE_NO_PROCESSING: // No processing active (Note: this state must always be present and left empty)
	            ;
	            
	        #FB_STATE_PROCESSING:
	            // Processing active
	            // 
	            #statRunTime := RUNTIME(MEM := #statMemStart);
	            
	            REPEAT
	                IF TypeOfDB(#statActDB_NUMBER) = LSimaHydTO_typeVCharData THEN
	                    // enter vchar to data exchange
	                    #tempInitDone := FALSE;
	                    FOR #tempInt := #statVCharArrMinIndex TO #statVCharArrMaxIndex DO
	                        IF #vCharArray[#tempInt].VChar_DB = #statActDB_NUMBER THEN
	                            #vCharArray[#tempInt].initialized := TRUE;
	                            #tempInitDone := TRUE;
	                            EXIT;
	                        END_IF;
	                    END_FOR;
	                    IF NOT #tempInitDone THEN
	                        FOR #tempInt := #statVCharArrMinIndex TO #statVCharArrMaxIndex DO
	                            IF NOT #vCharArray[#tempInt].initialized THEN
	                                #vCharArray[#tempInt].VChar_DB := #statActDB_NUMBER;
	                                #vCharArray[#tempInt].initialized := TRUE;
	                                #tempInitDone := TRUE;
	                                EXIT;
	                            END_IF;
	                            IF #tempInt = #statVCharArrMaxIndex THEN
	                                #statVCharArrayFull := TRUE;
	                            END_IF;
	                            
	                        END_FOR;
	                    END_IF;
	                    
	                ELSIF TypeOfDB(#statActDB_NUMBER) = LSimaHydTO_typeAxisData THEN
	                    #tempInitDone := FALSE;
	                    FOR #tempInt := #statAxesArrMinIndex TO #statAxesArrMaxIndex DO
	                        IF #axesArray[#tempInt].axisData = #statActDB_NUMBER THEN
	                            #axesArray[#tempInt].initialized := TRUE;
	                            #tempInitDone := TRUE;
	                            EXIT;
	                        END_IF;
	                    END_FOR;
	                    IF NOT #tempInitDone THEN
	                        FOR #tempInt := #statAxesArrMinIndex TO #statAxesArrMaxIndex DO
	                            IF NOT #axesArray[#tempInt].initialized THEN
	                                #axesArray[#tempInt].axisData := #statActDB_NUMBER;
	                                #axesArray[#tempInt].initialized := TRUE;
	                                #tempInitDone := TRUE;
	                                EXIT;
	                            END_IF;
	                            IF #tempInt = #statAxesArrMaxIndex THEN
	                                #statAxesArrayFull := TRUE;
	                            END_IF;
	                        END_FOR;
	                    END_IF;
	                    
	                END_IF;
	                IF #statAxesArrayFull AND #statVCharArrayFull THEN
	                    #statBusy := FALSE;
	                    #statStatus := #STATUS_EXECUTION_FINISHED;
	                END_IF;
	                
	                IF #statStatus = #STATUS_SUBSEQUENT_CALL THEN
	                    IF #statActDB_NUMBER < uint#65_535 THEN
	                        #statActDB_NUMBER += 1;
	                    ELSE
	                        #statBusy := FALSE;
	                        #statStatus := #STATUS_EXECUTION_FINISHED;
	                    END_IF;
	                END_IF;
	                #statMem := #statMemStart;
	                #statRunTime := RUNTIME(MEM := #statMem);
	            UNTIL NOT #statBusy OR #statRunTime > 0.01 // interupt after 10 ms
	            END_REPEAT;
	            
	            
	        ELSE // Undefined state in state machine reached
	            #statStatus := #ERR_UNDEFINED_STATE;
	    END_CASE;
	END_REGION STATE_MACHINE
	
	REGION OUTPUTS
	    // Write outputs
	    IF (#statStatus = #STATUS_EXECUTION_FINISHED) AND (#statDone = FALSE) THEN // Execution finished without errors
	        #statDone := TRUE;
	        #statBusy := FALSE;
	        #statError := FALSE;
	        #statFBState := #FB_STATE_NO_PROCESSING; // Switch state machine to "no processing"
	        
	    ELSIF (#statStatus.%X15 = TRUE) AND (#statError = FALSE) THEN // Error occurred (#statStatus is 16#8000 to 16#FFFF)
	        #statDone := FALSE;
	        #statBusy := FALSE;
	        #statError := TRUE;
	        #statFBState := #FB_STATE_NO_PROCESSING; // Switch state machine to "no processing"
	        
	    ELSIF (#tempExecute = FALSE) AND ((#statDone = TRUE) OR (#statError = TRUE)) THEN // Reset outputs
	        #statDone := FALSE;
	        #statBusy := FALSE;
	        #statError := FALSE;
	        #statStatus := #STATUS_NO_CALL;
	    END_IF;
	    
	    // Write static values to outputs
	    #done := #statDone;
	    #busy := #statBusy;
	    #error := #statError;
	    #status := #statStatus;
	END_REGION OUTPUTS
END_FUNCTION_BLOCK

FUNCTION_BLOCK "SimaHydTO_VCharManagement"
{ S7_Optimized_Access := 'TRUE' }
FAMILY : SimaHydTO
VERSION : 1.0
   VAR_IN_OUT 
      hmiConnection : "SimaHydTO_typeHMIConnection";
      axisData : "LSimaHydTO_typeAxisData";
      vCharArray : Array[*] of "SimaHydTO_typeVCharArray";
   END_VAR

   VAR 
      statSaveDBL { ExternalAccessible := 'False'; ExternalVisible := 'False'; ExternalWritable := 'False'} : Bool;
      statLoadDBL { ExternalAccessible := 'False'; ExternalVisible := 'False'; ExternalWritable := 'False'} : Bool;
      statEditOld { ExternalAccessible := 'False'; ExternalVisible := 'False'; ExternalWritable := 'False'} : Bool;
      statActivateOld { ExternalAccessible := 'False'; ExternalVisible := 'False'; ExternalWritable := 'False'} : Bool;
      statAbortOld { ExternalAccessible := 'False'; ExternalVisible := 'False'; ExternalWritable := 'False'} : Bool;
      statRestoreOld { ExternalAccessible := 'False'; ExternalVisible := 'False'; ExternalWritable := 'False'} : Bool;
      statApplayOld { ExternalAccessible := 'False'; ExternalVisible := 'False'; ExternalWritable := 'False'} : Bool;
      statDefaultAxisData { ExternalAccessible := 'False'; ExternalVisible := 'False'; ExternalWritable := 'False'} : "SimaHydTO_typeHMIConnectionParameterSettingsAxisData";
      instMC_WriteToROM { ExternalAccessible := 'False'; ExternalVisible := 'False'; ExternalWritable := 'False'} : "LSimaHydTO_MC_WriteToROM";
      instMC_ReadFromROM { ExternalAccessible := 'False'; ExternalVisible := 'False'; ExternalWritable := 'False'} : "LSimaHydTO_MC_ReadFromROM";
      instVCharSelector { ExternalAccessible := 'False'; ExternalVisible := 'False'; ExternalWritable := 'False'} : "SimaHydTO_HmiVCharSelector";
      statSaveOld { ExternalAccessible := 'False'; ExternalVisible := 'False'; ExternalWritable := 'False'} : Bool;
   END_VAR

   VAR_TEMP 
      tempVariant : Variant;
      tempErrorVariant : Int;
      tempDbAny : DB_ANY;
      tempVCharData : REF_TO "LSimaHydTO_typeVCharData";
   END_VAR


BEGIN
	//=============================================================================
	//SIEMENS AG
	//(c)Copyright 2016 All Rights Reserved
	//-----------------------------------------------------------------------------
	//Library:       SimaHydTO_VCharManagement
	//Tested with:   S7-1500 V2.5
	//Engineering:   TIA Portal V15
	//Restrictions:  -
	//Requirements:  S7-1500(T)
	//Functionality: Manipulate active VChar of selected hydraulic axis
	//-----------------------------------------------------------------------------
	//Change log table:
	//Version  Date       Expert in charge Changes applied
	//01.00.00 17.07.2019 ArSc             First released version
	//=============================================================================
	
	  // Vchar selection
	  #instVCharSelector(command:=#hmiConnection.ParameterSettings.Commands.VCharSelector,
	                       status:=#hmiConnection.ParameterSettings.Status.VCharSelector,
	                       vCharArray:=#vCharArray);
	  
	  
	  IF #hmiConnection.ParameterSettings.Commands.ApplyVChar
	    AND NOT #statApplayOld
	    AND #hmiConnection.ParameterSettings.Status.VCharSelector.dataValid
	  THEN
	    #axisData.ValveCharacteristic.DB_NUMBER := #hmiConnection.ParameterSettings.Status.VCharSelector.selectedVChar;
	    #hmiConnection.AxisSelector.Status.selectedVChar := #hmiConnection.ParameterSettings.Status.VCharSelector.selectedVChar;
	    #hmiConnection.AxisSelector.Status.selectedVCharInteger := DB_ANY_TO_UINT(#hmiConnection.ParameterSettings.Status.VCharSelector.selectedVChar);
	    
	    
	    #hmiConnection.ParameterSettings.AxisData.VCharName := #hmiConnection.ParameterSettings.Status.VCharSelector.selectedVCharName;
	    #hmiConnection.ParameterSettings.AxisData.ValveCharacteristic.DB_NUMBER := #hmiConnection.ParameterSettings.Status.VCharSelector.selectedVChar;
	    
	    #hmiConnection.AxisSelector.Status.selectedVCharName := #hmiConnection.ParameterSettings.Status.VCharSelector.selectedVCharName;
	    
	    
	    
	  END_IF;
	
	#statApplayOld := #hmiConnection.ParameterSettings.Commands.ApplyVChar;
	
END_FUNCTION_BLOCK

FUNCTION "SimaHydTO_GetAxisToUnits_PosAxis" : "SimaHydTO_typeHMIConnectionAxisToDataAxisUnits"
{ S7_Optimized_Access := 'TRUE' }
FAMILY : SimaHydTO
VERSION : 1.0
   VAR_INPUT 
      axisTO {InstructionName := 'TO_PositioningAxis'; LibVersion := '4.0'} : TO_PositioningAxis;
   END_VAR


BEGIN
	//=============================================================================
	//SIEMENS AG
	//(c)Copyright 2016 All Rights Reserved
	//-----------------------------------------------------------------------------
	//Library:       SimaHyd_AxisBasics
	//Tested with:   S7-1500 V2.5
	//Engineering:   TIA Portal V15
	//Restrictions:  Motion Control Library V4.0
	//Requirements:  S7-1500(T)
	//Functionality: Get axis units of TO_PositioningAxis
	//-----------------------------------------------------------------------------
	//Change log table:
	//Version  Date       Expert in charge Changes applied
	//01.00.00 20.05.2019 ArSc             First released version
	//=============================================================================
	
	
	//-----------------------------------------------------------------------------
	//Write axis units
	//-----------------------------------------------------------------------------
	
	#SimaHydTO_GetAxisToUnits_PosAxis.forceUnit := #axisTO.Units.ForceUnit;
	#SimaHydTO_GetAxisToUnits_PosAxis.lengthUnit := #axisTO.Units.LengthUnit;
	#SimaHydTO_GetAxisToUnits_PosAxis.velocityUnit := #axisTO.Units.VelocityUnit;
	
END_FUNCTION

FUNCTION "SimaHydTO_GetAxisToUnits_SyncAxis" : "SimaHydTO_typeHMIConnectionAxisToDataAxisUnits"
{ S7_Optimized_Access := 'TRUE' }
FAMILY : SimaHydTO
VERSION : 1.0
   VAR_INPUT 
      axisTO {InstructionName := 'TO_SynchronousAxis'; LibVersion := '4.0'} : TO_SynchronousAxis;
   END_VAR


BEGIN
	//=============================================================================
	//SIEMENS AG
	//(c)Copyright 2016 All Rights Reserved
	//-----------------------------------------------------------------------------
	//Library:       SimaHyd_AxisBasics
	//Tested with:   S7-1500 V2.5
	//Engineering:   TIA Portal V15
	//Restrictions:  Motion Control Library V4.0
	//Requirements:  S7-1500(T)
	//Functionality: Get axis units of TO_SynchronousAxis
	//-----------------------------------------------------------------------------
	//Change log table:
	//Version  Date       Expert in charge Changes applied
	//01.00.00 20.05.2019 ArSc             First released version
	//=============================================================================
	
	
	//-----------------------------------------------------------------------------
	//Write axis data
	//-----------------------------------------------------------------------------
	#SimaHydTO_GetAxisToUnits_SyncAxis := "SimaHydTO_GetAxisToUnits_PosAxis"(#axisTO);
END_FUNCTION

FUNCTION "SimaHydTO_HmiAxisAnimation" : Void
{ S7_Optimized_Access := 'TRUE' }
FAMILY : SimaHydTO
VERSION : 1.0
   VAR_IN_OUT 
      hmiConnection : "SimaHydTO_typeHMIConnection";
      axisData : "LSimaHydTO_typeAxisData";
   END_VAR

   VAR_TEMP 
      tempPositionLimitsSW : "LSimaHydTO_typePositionLimits";
      tempTravelDistance : LReal;
   END_VAR


BEGIN
	//=============================================================================
	//SIEMENS AG
	//(c)Copyright 2016 All Rights Reserved
	//-----------------------------------------------------------------------------
	//Library:       SimaHydTO_HMI
	//Tested with:   S7-1500 V2.5
	//Engineering:   TIA Portal V15
	//Restrictions:  -
	//Requirements:  S7-1500(T)
	//Functionality: Transfer data from/to HMI to/from selected axis
	//-----------------------------------------------------------------------------
	//Change log table:
	//Version  Date       Expert in charge Changes applied
	//01.00.00 12.07.2019 ArSc             First released version
	//=============================================================================
	
	
	// 
	IF #hmiConnection.AxisSelector.Status.dataValid 
	THEN
	  //Read data
	  //Check data
	  IF #axisData.DataInitialized = TRUE
	  THEN
	    //Calculate HMI data
	    #tempPositionLimitsSW := #axisData.Internal.PositionLimits_SW;
	    IF (#tempPositionLimitsSW.Active = True)
	    THEN
	      #hmiConnection.HmiData.MinPosition := #tempPositionLimitsSW.MinPosition;
	      #hmiConnection.HmiData.MaxPosition := #tempPositionLimitsSW.MaxPosition;
	      #tempTravelDistance := (#tempPositionLimitsSW.MaxPosition - #tempPositionLimitsSW.MinPosition);
	      //Calculate percent value
	      IF (#tempTravelDistance > 0.0)
	      THEN
	        #hmiConnection.HmiData.ActualPositionPercent := DINT_TO_INT(TRUNC(100.0 * ((#axisData.ActualPosition - #tempPositionLimitsSW.MinPosition) /
	                                                            #tempTravelDistance)));
	        
	        #hmiConnection.HmiData.SafetyDistanceAnimation := #tempPositionLimitsSW.MinPosition + #hmiConnection.BasicAxisControl.ControlDirectOutput.safetyDistance;
	
	    
	
	      ELSE
	          #hmiConnection.HmiData.ActualPositionPercent := 0;
	          #hmiConnection.HmiData.SafetyDistanceAnimation := 0.0;
	      END_IF;
	    ELSE
	      #hmiConnection.HmiData.MinPosition := 0.0;
	      #hmiConnection.HmiData.MaxPosition := 0.0;
	      #hmiConnection.HmiData.ActualPositionPercent := 0;
	      #hmiConnection.HmiData.SafetyDistanceAnimation := 0.0;
	      #hmiConnection.HmiData.selectedAxis := 0;
	      #hmiConnection.HmiData.selectedAxisTO := 0;
	    END_IF;
	  END_IF;
	  #hmiConnection.AxisData.Force := #axisData.Force;
	  #hmiConnection.AxisData.Velocity := #axisData.Velocity;
	  #hmiConnection.AxisData.Position := #axisData.Position;
	  #hmiConnection.AxisData.ActualForce := #axisData.ActualForce;
	  #hmiConnection.AxisData.ActualVelocity := #axisData.ActualVelocity;
	  #hmiConnection.AxisData.ActualPosition := #axisData.ActualPosition;
	  #hmiConnection.AxisData.Status_A_Transducer.PressureValue := #axisData.Status_A_Transducer.PressureValue;
	  #hmiConnection.AxisData.Status_B_Transducer.PressureValue := #axisData.Status_B_Transducer.PressureValue;
	  #hmiConnection.AxisData.StatusActor := #axisData.StatusActor;
	  
	END_IF;
	
END_FUNCTION

FUNCTION "LSimaHydTO_AreaToDiameter" : Void
{ S7_Optimized_Access := 'TRUE' }
AUTHOR : APC_ERLF
FAMILY : LSimaHydTO
VERSION : 1.0
   VAR_INPUT 
      pistonArea : LReal;
      pistonRodArea : LReal;
   END_VAR

   VAR_OUTPUT 
      pistonDiameter : LReal;
      pistonRodDiameter : LReal;
   END_VAR


BEGIN
	//================================================================================
	//SIEMENS AG // (c)Copyright 2019 All Rights Reserved
	//--------------------------------------------------------------------------------
	//Library:       LSimaHydTO
	//Tested with:   S7-15xx
	//Engineering:   TIA Portal  V15
	//Restrictions:  -
	//Requirements:  S7-1500 (FW 2.5)
	//Functionality: HMI support program - Internal use  
	//
	//--------------------------------------------------------------------------------
	//Change log table:
	//
	//Version     Date          Expert in charge    Changes applied
	//01.00.00    15.03.2018    APC_ERLF            First released version
	//================================================================================
	
	
	IF #pistonArea > 0.0 THEN
	  #pistonDiameter := SQRT(#pistonArea * 1.2732395);
	  IF #pistonRodArea > 0.0 AND #pistonRodArea < #pistonArea THEN
	    #pistonRodDiameter := SQRT(#pistonDiameter*#pistonDiameter -  #pistonRodArea * 1.2732395);
	  ELSE
	    #pistonRodDiameter := 0.0;
	  END_IF;
	ELSE
	  #pistonRodDiameter := 0.0;
	  #pistonDiameter := 0.0;
	END_IF;
	
	
END_FUNCTION

FUNCTION "LSimaHydTO_Covariance" : Int
{ S7_Optimized_Access := 'TRUE' }
AUTHOR : APC_ERLF
FAMILY : LSimaHydTO
VERSION : 1.0
   VAR_INPUT 
      firstIdx : Int;
      numOfPoints : Int;
   END_VAR

   VAR_OUTPUT 
      factor : Real;
      correlation : Real;
   END_VAR

   VAR_IN_OUT 
      valuesX : Array[*] of Real;
      valuesY : Array[*] of Real;
   END_VAR

   VAR_TEMP 
      i : Int;
      ret : Int;
      sum2X : Real;
      sum2Y : Real;
      meanValueX : Real;
      meanValueY : Real;
      sumX : Real;
      sumY : Real;
      varianceX : Real;
      variancey : Real;
      sumCoVar : Real;
      covariance : Real;
      tempLB : Int;
      tempUB : Int;
      lastIdx : Int;
   END_VAR


BEGIN
	//================================================================================
	//SIEMENS AG // (c)Copyright 2019 All Rights Reserved
	//--------------------------------------------------------------------------------
	//Library:       LSimaHydTO
	//Tested with:   S7-15xx
	//Engineering:   TIA Portal  V15
	//Restrictions:  -
	//Requirements:  S7-1500 (FW 2.5)
	//Functionality: HMI support program - Internal use  
	//
	//--------------------------------------------------------------------------------
	//Change log table:
	//
	//Version     Date          Expert in charge    Changes applied
	//01.00.00    15.03.2018    APC_ERLF            First released version
	//================================================================================
	
	
	IF #numOfPoints < 2 THEN
	  #LSimaHydTO_Covariance := -1;
	  RETURN;
	END_IF;
	#tempLB := DINT_TO_INT(MAX(IN1 := LOWER_BOUND(ARR:=#valuesX, DIM:=1),IN2 := LOWER_BOUND(ARR:=#valuesY, DIM:=1)));
	#tempUB := DINT_TO_INT(MIN(IN1 := UPPER_BOUND(ARR := #valuesX, DIM := 1), IN2 := UPPER_BOUND(ARR := #valuesY, DIM := 1)));
	#lastIdx := #firstIdx + #numOfPoints - 1;
	IF #tempLB > #firstIdx  THEN
	  #ret := -2;
	ELSIF #tempUB < #lastIdx THEN
	  #ret := -3;
	ELSE
	  #ret := 0;
	  #sumX := 0.0;
	  #sumY := 0.0;
	  #sum2X := 0.0;
	  #sum2Y := 0.0;
	  #sumCoVar := 0.0;
	  FOR #i := #firstIdx TO #lastIdx DO
	    #sumX := #sumX + #valuesX[#i];
	    #sumY := #sumY + #valuesY[#i];
	  END_FOR;
	  #meanValueX := #sumX / #numOfPoints;
	  #meanValueY := #sumY / #numOfPoints;
	  FOR #i := #firstIdx TO #lastIdx DO
	    #sum2X := #sum2X + SQR(#valuesX[#i] - #meanValueX);
	    #sum2Y := #sum2Y + SQR(#valuesY[#i] - #meanValueY);
	    #sumCoVar := #sumCoVar + (#valuesX[#i] - #meanValueX) * (#valuesY[#i] - #meanValueY);
	  END_FOR;
	  #varianceX := #sum2X / (#numOfPoints - 1);
	  #variancey := #sum2Y / (#numOfPoints - 1);
	  #covariance := #sumCoVar / (#numOfPoints - 1);
	  #factor := #covariance / #varianceX;
	  #correlation := #covariance / (SQRT(#varianceX) * SQRT(#variancey));
	END_IF;
	#LSimaHydTO_Covariance := #ret;
	
	
END_FUNCTION

FUNCTION "LSimaHydTO_DiameterToArea" : Void
{ S7_Optimized_Access := 'TRUE' }
AUTHOR : APC_ERLF
FAMILY : LSimaHydTO
VERSION : 1.0
   VAR_INPUT 
      pistonDiameter : LReal;
      pistonRodDiameter : LReal;
   END_VAR

   VAR_OUTPUT 
      pistonArea : LReal;
      pistonRodArea : LReal;
   END_VAR


BEGIN
	//================================================================================
	//SIEMENS AG // (c)Copyright 2019 All Rights Reserved
	//--------------------------------------------------------------------------------
	//Library:       LSimaHydTO
	//Tested with:   S7-15xx
	//Engineering:   TIA Portal  V15
	//Restrictions:  -
	//Requirements:  S7-1500 (FW 2.5)
	//Functionality: HMI support program - Internal use  
	//
	//--------------------------------------------------------------------------------
	//Change log table:
	//
	//Version     Date          Expert in charge    Changes applied
	//01.00.00    15.03.2018    APC_ERLF            First released version
	//================================================================================
	
	
	IF #pistonDiameter > 0.0 THEN
	  #pistonArea := #pistonDiameter*#pistonDiameter * 0.7853981;
	  IF #pistonRodDiameter > 0.0 AND #pistonRodDiameter < #pistonDiameter THEN
	    #pistonRodArea := (#pistonDiameter*#pistonDiameter -  #pistonRodDiameter*#pistonRodDiameter) * 0.7853981;
	  ELSE
	    #pistonRodArea := 0.0;
	  END_IF;
	ELSE
	  #pistonRodArea := 0.0;
	  #pistonArea := 0.0;
	END_IF;
	
	
END_FUNCTION

FUNCTION "LSimaHydTO_GetAxisForceCommandState" : Word
{ S7_Optimized_Access := 'TRUE' }
AUTHOR : APC_ERLF
FAMILY : LSimaHydTO
VERSION : 1.0
   VAR_INPUT 
      commandID : UDInt;
   END_VAR

   VAR_IN_OUT 
      axis : "LSimaHydTO_typeAxisData";
   END_VAR

   VAR_TEMP 
      tempRetVal : Word;
   END_VAR

   VAR CONSTANT 
      MOTION_STATE_NOT_EXISTEND : Word := 16#0000;
      MOTION_STATE_BUFFERED_OR_MOTION : Word := 16#0001;
      MOTION_STATE_EXECUTED : Word := 16#0010;
      MOTION_STATE_ABORTED : Word := 16#0020;
      MOTION_STATE_ERROR : Word := 16#8000;
   END_VAR


BEGIN
	//================================================================================
	//SIEMENS AG // (c)Copyright 2019 All Rights Reserved
	//--------------------------------------------------------------------------------
	//Library:       LSimaHydTO
	//Tested with:   S7-15xx
	//Engineering:   TIA Portal  V15
	//Restrictions:  -
	//Requirements:  S7-1500 (FW 2.5)
	//Functionality: - for internal use
	//
	//--------------------------------------------------------------------------------
	//Change log table:
	//
	//Version     Date          Expert in charge    Changes applied
	//01.00.00    15.03.2018    APC_ERLF            First released version
	//================================================================================
	
	
	IF #axis.Internal.Control.ForceCommand.commandID = #commandID THEN
	  #tempRetVal := #MOTION_STATE_BUFFERED_OR_MOTION;
	ELSIF #axis.Internal.MotionData.ForceCmdTracking.CommandID = #commandID THEN
	  IF (#axis.Internal.MotionData.ForceCmdTracking.State AND #MOTION_STATE_BUFFERED_OR_MOTION) <> 0 THEN
	    #tempRetVal := #MOTION_STATE_BUFFERED_OR_MOTION;
	  ELSE
	    #tempRetVal := #axis.Internal.MotionData.ForceCmdTracking.State;
	  END_IF;
	ELSE
	  #tempRetVal := #MOTION_STATE_NOT_EXISTEND;
	END_IF;
	#LSimaHydTO_GetAxisForceCommandState := #tempRetVal;
	
	
END_FUNCTION

FUNCTION "LSimaHydTO_GetCommandID" : UDInt
{ S7_Optimized_Access := 'TRUE' }
AUTHOR : APC_ERLF
FAMILY : LSimaHydTO
VERSION : 1.0
   VAR_IN_OUT 
      axis : "LSimaHydTO_typeAxisData";
   END_VAR


BEGIN
	//================================================================================
	//SIEMENS AG // (c)Copyright 2019 All Rights Reserved
	//--------------------------------------------------------------------------------
	//Library:       LSimaHydTO
	//Tested with:   S7-15xx
	//Engineering:   TIA Portal  V15
	//Restrictions:  -
	//Requirements:  S7-1500 (FW 2.5)
	//Functionality: - for internal use
	//
	//--------------------------------------------------------------------------------
	//Change log table:
	//
	//Version     Date          Expert in charge    Changes applied
	//01.00.00    15.03.2018    APC_ERLF            First released version
	//================================================================================
	
	
	#axis.Internal.CommandIDPool := #axis.Internal.CommandIDPool+1;
	IF #axis.Internal.CommandIDPool = 0 THEN
	  #axis.Internal.CommandIDPool := #axis.Internal.CommandIDPool + 1;
	END_IF;
	#LSimaHydTO_GetCommandID:= #axis.Internal.CommandIDPool;
	
	
END_FUNCTION

FUNCTION "LSimaHydTO_GetPosAxisData" : Void
{ S7_Optimized_Access := 'TRUE' }
AUTHOR : APC_ERLF
FAMILY : LSimaHydTO
VERSION : 1.0
   VAR_INPUT 
      axisTO {InstructionName := 'TO_PositioningAxis'; LibVersion := '4.0'} : TO_PositioningAxis;
   END_VAR

   VAR_OUTPUT 
      statusWord : DWord;
      errorWord : DWord;
      errorDetail : "LSimaHydTO_typeErrorDetail";
      velocity : LReal;
      acceleration : LReal;
      position : LReal;
      actualSpeed : LReal;
      actualVelocity : LReal;
      actualAcceleration : LReal;
      actualPosition : LReal;
      referenceSpeed : LReal;
      positionLimits_SW {InstructionName := 'TO_Struct_PositionLimitsSW'; LibVersion := '4.0'} : TO_Struct_PositionLimitsSW;
      dynamicLimits : "LSimaHydTO_typeDynamicLimits";
   END_VAR


BEGIN
	//================================================================================
	//SIEMENS AG // (c)Copyright 2019 All Rights Reserved
	//--------------------------------------------------------------------------------
	//Library:       LSimaHydTO
	//Tested with:   S7-15xx
	//Engineering:   TIA Portal  V15
	//Restrictions:  -
	//Requirements:  S7-1500 (FW 2.5)
	//Functionality: - for internal use
	//
	//--------------------------------------------------------------------------------
	//Change log table:
	//
	//Version     Date          Expert in charge    Changes applied
	//01.00.00    15.03.2018    APC_ERLF            First released version
	//================================================================================
	
	#statusWord := #axisTO.StatusWord;
	#errorWord := #axisTO.ErrorWord;
	#velocity := #axisTO.Velocity;
	#acceleration := #axisTO.Acceleration;
	#position := #axisTO.Position;
	#actualSpeed := #axisTO.ActualSpeed;
	#actualVelocity := #axisTO.ActualVelocity;
	#actualAcceleration := #axisTO.#ActualAcceleration;
	#actualPosition := #axisTO.ActualPosition;
	#referenceSpeed := #axisTO.Actor.DriveParameter.ReferenceSpeed;
	#errorDetail.Number := #axisTO.ErrorDetail.Number;
	#errorDetail.Reaction := #axisTO.ErrorDetail.Reaction;
	//software limit switches
	#positionLimits_SW.Active := #axisTO.PositionLimits_SW.Active;
	#positionLimits_SW.MaxPosition := #axisTO.PositionLimits_SW.MaxPosition;
	#positionLimits_SW.MinPosition := #axisTO.PositionLimits_SW.MinPosition;
	#dynamicLimits.MaxVelocity := MIN(IN1 := #axisTO.DynamicLimits.MaxVelocity, IN2 := #axisTO.DynamicLimits.Velocity);
	#dynamicLimits.MaxAcceleration := #axisTO.DynamicLimits.MaxAcceleration;
	#dynamicLimits.MaxDeceleration := #axisTO.DynamicLimits.MaxDeceleration;
	#dynamicLimits.MaxJerk := #axisTO.DynamicLimits.MaxJerk;
	
	
END_FUNCTION

FUNCTION_BLOCK "LSimaHydTO_HandleDBL"
{ S7_Optimized_Access := 'TRUE' }
AUTHOR : APC_ERLF
FAMILY : LSimaHydTO
VERSION : 1.0
   VAR_INPUT 
      executeRead : Bool;
      executeWrite : Bool;
   END_VAR

   VAR_OUTPUT 
      busy { ExternalWritable := 'False'} : Bool;
      done { ExternalWritable := 'False'} : Bool;
      error { ExternalWritable := 'False'} : Bool;
      errorID { ExternalWritable := 'False'} : Int;
   END_VAR

   VAR_IN_OUT 
      memoryDB : Variant;
      cardDB : Variant;
   END_VAR

   VAR 
      statFBState { ExternalAccessible := 'False'; ExternalVisible := 'False'; ExternalWritable := 'False'} : Int;
      statExecuteReadOld { ExternalAccessible := 'False'; ExternalVisible := 'False'; ExternalWritable := 'False'} : Bool;
      statExecuteWriteOld { ExternalAccessible := 'False'; ExternalVisible := 'False'; ExternalWritable := 'False'} : Bool;
      statRetVal { ExternalAccessible := 'False'; ExternalVisible := 'False'; ExternalWritable := 'False'} : Int;
   END_VAR

   VAR CONSTANT 
      FB_STATE_IDLE : Int;
      FB_STATE_READ : Int := 10;
      FB_STATE_WRITE : Int := 20;
      FB_STATE_ERROR : Int := 100;
   END_VAR


BEGIN
	//================================================================================
	//SIEMENS AG // (c)Copyright 2019 All Rights Reserved
	//--------------------------------------------------------------------------------
	//Library:       LSimaHydTO
	//Tested with:   S7-15xx
	//Engineering:   TIA Portal  V15 (SW 2.5)
	//Restrictions:  -
	//Requirements:  S7-1500
	//Functionality: Save and load DB data to/from card
	//
	//--------------------------------------------------------------------------------
	//Change log table:
	//
	//Version     Date          Expert in charge    Changes applied
	//01.00.00    15.03.2018    APC_ERLF            First released version
	//================================================================================
	
	
	CASE #statFBState OF
	    
	  #FB_STATE_IDLE: 
	
	    IF #executeRead AND NOT #statExecuteReadOld THEN
	      #busy := false;
	      #done := false;
	      #error := false;
	      #errorID := 0;
	      #statRetVal := READ_DBL(REQ := #executeRead, SRCBLK := #cardDB, BUSY => #busy, DSTBLK => #memoryDB);
	      IF #busy THEN
	        #statFBState := #FB_STATE_READ;
	      ELSE
	        #error := TRUE;
	        #errorID := #statRetVal;
	        #statFBState := #FB_STATE_ERROR;
	      END_IF;
	    ELSIF  #executeWrite AND NOT #statExecuteWriteOld THEN
	      #busy := false;
	      #done := false;
	      #error := false;
	      #errorID := 0;
	      #statRetVal := WRIT_DBL(REQ := #executeWrite, SRCBLK :=#memoryDB , BUSY => #busy, DSTBLK => #cardDB);
	      IF #busy THEN
	        #statFBState := #FB_STATE_WRITE;
	      ELSE
	        #error := TRUE;
	        #errorID := #statRetVal;
	        #statFBState := #FB_STATE_ERROR;
	      END_IF;
	    ELSIF NOT(#executeRead OR #executeWrite) THEN
	      #done := FALSE;
	      #busy := FALSE;
	    END_IF;
	    
	    
	  #FB_STATE_READ:
	    
	    #statRetVal := READ_DBL(REQ := #executeRead, SRCBLK := #cardDB, BUSY => #busy, DSTBLK => #memoryDB);;
	    IF NOT #busy THEN
	      IF #statRetVal = 0 THEN
	        #done := TRUE;
	        #statFBState := #FB_STATE_IDLE;
	      ELSE
	        #error := TRUE;
	        #errorID := #statRetVal;
	        #statFBState := #FB_STATE_ERROR;
	      END_IF;
	    END_IF;
	    
	    
	  #FB_STATE_WRITE:
	    
	    #statRetVal := WRIT_DBL(REQ := #executeWrite, SRCBLK :=#memoryDB , BUSY => #busy, DSTBLK => #cardDB);
	    IF NOT #busy THEN
	      IF #statRetVal = 0 THEN
	        #done := TRUE;
	        #statFBState := #FB_STATE_IDLE;
	      ELSE
	        #error := TRUE;
	        #errorID := #statRetVal;
	        #statFBState := #FB_STATE_ERROR;
	      END_IF;
	    END_IF;
	    
	    
	  #FB_STATE_ERROR:
	    
	    IF NOT (#executeRead OR #executeWrite) THEN
	      #statFBState := #FB_STATE_IDLE;
	    END_IF;
	  ELSE
	    ;
	END_CASE;
	
	#statExecuteReadOld := #executeRead;
	#statExecuteWriteOld := #executeWrite;
	
	
END_FUNCTION_BLOCK

FUNCTION_BLOCK "LSimaHydTO_MC_ForceControl"
{ S7_Optimized_Access := 'TRUE' }
AUTHOR : APC_ERLF
FAMILY : LSimaHydTO
VERSION : 1.0
   VAR_INPUT 
      execute : Bool;
      forceControlProfile : UInt;
      mode : DInt;
      forceProfileMode : DInt;
      conditionMode : DInt := 1;
      compareMode : DInt := 1;
      conditionValue : LReal;
      forceValue : LReal;
      forceDerivedValue : LReal;
      velocityLimitingValue : LReal;
   END_VAR

   VAR_OUTPUT 
      done { ExternalWritable := 'False'} : Bool;
      inForceControl { ExternalWritable := 'False'} : Bool;
      busy { ExternalWritable := 'False'} : Bool;
      commandAborted { ExternalWritable := 'False'} : Bool;
      error { ExternalWritable := 'False'} : Bool;
      errorID { ExternalWritable := 'False'} : Word;
   END_VAR

   VAR_IN_OUT 
      axis : "LSimaHydTO_typeAxisData";
   END_VAR

   VAR 
      statFBState { ExternalAccessible := 'False'; ExternalVisible := 'False'; ExternalWritable := 'False'} : DInt;
      statCommandID { ExternalAccessible := 'False'; ExternalVisible := 'False'; ExternalWritable := 'False'} : UDInt;
      statCmdState { ExternalAccessible := 'False'; ExternalVisible := 'False'; ExternalWritable := 'False'} : Word;
      statExecuteOld { ExternalAccessible := 'False'; ExternalVisible := 'False'; ExternalWritable := 'False'} : Bool;
   END_VAR

   VAR CONSTANT 
      NO_ERROR : Word := 16#0000;
      STATE_IDLE : DInt;
      STATE_FIRST_CYCLE : DInt := 10;
      STATE_BUSY : DInt := 20;
      STATE_DONE : DInt := 30;
      STATE_COMMAND_ABORTED : DInt := 40;
      STATE_ERROR : DInt := 100;
      MOTION_STATE_NOT_EXISTEND : Word := 16#0000;
      MOTION_STATE_BUFFERED_OR_MOTION : Word := 16#0001;
      MOTION_STATE_EXECUTED : Word := 16#0010;
      MOTION_STATE_ABORTED : Word := 16#0020;
      MOTION_STATE_ERROR : Word := 16#8000;
      NO_ERROR_REACTION : DInt := 0;
      ALARM_AXIS_ERROR_OCCURED : Word := 16#8001;
      ALARM_WRONG_MODE : Word := 16#800A;
      ALARM_AXIS_DISABLED : Word := 16#800F;
      ALARM_FORCE_PROFILE_MODE : Word := 16#80B1;
      ALARM_CONDITION_MODE : Word := 16#80B2;
      ALARM_FORCE_PROFILE : Word := 16#80B3;
      ALARM_COMPARE_MODE : Word := 16#80B4;
      ALARM_FORCE_DERIVED_VALUE : Word := 16#80B5;
   END_VAR


BEGIN
	//================================================================================
	//SIEMENS AG // (c)Copyright 2019 All Rights Reserved
	//--------------------------------------------------------------------------------
	//Library:       LSimaHydTO
	//Tested with:   S7-15xx
	//Engineering:   TIA Portal  V15
	//Restrictions:  -
	//Requirements:  S7-1500 (FW 2.5)
	//Functionality: Function to activate and deactivate pressure control mode for an axis.
	//               In addition, you can specify the conditions under which pressure
	//               control becomes active.
	//
	//--------------------------------------------------------------------------------
	//Change log table:
	//
	//Version     Date          Expert in charge    Changes applied
	//01.00.00    15.03.2018    APC_ERLF            First released version
	//================================================================================
	
	
	//----------------------------------------------------------------------
	//start
	//----------------------------------------------------------------------
	
	//rising edge of execute starts functionality
	IF #execute AND NOT #statExecuteOld THEN
	  //initialization
	  #done := FALSE;
	  #commandAborted := FALSE;
	  #inForceControl := FALSE;
	  #busy := FALSE;
	  #error := FALSE;
	  #errorID := #NO_ERROR;
	  #statFBState := #STATE_FIRST_CYCLE;
	END_IF;
	
	
	//----------------------------------------------------------------------
	//busy
	//----------------------------------------------------------------------
	
	CASE #statFBState OF
	    
	  #STATE_FIRST_CYCLE:
	    
	    //==================================================================
	    //This state runs just one time after a rising edge on execute and
	    //calls the function to start the motion.
	    //Get a commandId and buffer it for tracking the command in the
	    //following state STATE_BUSY
	    //==================================================================
	    
	    #commandAborted := FALSE;
	    IF #mode < 0 OR #mode > 2 THEN
	      #error := TRUE;
	      #errorID := #ALARM_WRONG_MODE;
	      #statFBState := #STATE_ERROR;
	    ELSIF #mode <> 0 AND (#forceProfileMode < 0 OR #forceProfileMode > 2) THEN
	      #error := TRUE;
	      #errorID := #ALARM_FORCE_PROFILE_MODE;
	      #statFBState := #STATE_ERROR;
	    ELSIF #mode = 2 AND (#conditionMode < 1 OR #conditionMode > 3) THEN
	      #error := TRUE;
	      #errorID := #ALARM_CONDITION_MODE;
	      #statFBState := #STATE_ERROR;
	    ELSIF #mode = 2 AND #conditionMode > 1 AND (#compareMode < 1 OR #compareMode > 2) THEN
	      #error := TRUE;
	      #errorID := #ALARM_COMPARE_MODE;
	      #statFBState := #STATE_ERROR;
	    ELSIF #mode > 0 AND #forceProfileMode = 0 AND #forceDerivedValue <= 0.0 THEN
	      #error := TRUE;
	      #errorID := #ALARM_FORCE_DERIVED_VALUE;
	      #statFBState := #STATE_ERROR;
	    ELSIF NOT #axis.StatusActor.Enabled THEN
	      #error := TRUE;
	      #errorID := #ALARM_AXIS_DISABLED;
	      #statFBState := #STATE_ERROR;
	    ELSIF #axis.#ErrorWord <> 0 AND #axis.ErrorDetail.Reaction <> #NO_ERROR_REACTION THEN
	      #error := TRUE;
	      #errorID := #ALARM_AXIS_ERROR_OCCURED;
	      #statFBState := #STATE_ERROR;
	    ELSE
	      IF #mode <> 0 AND #forceProfileMode > 0 THEN
	        //check force profile DB 
	        IF #forceControlProfile > 0 THEN
	          #axis.StatusForceProfile.ActualProfile := #forceControlProfile;
	        ELSE
	          #axis.StatusForceProfile.ActualProfile := 0;
	          #error := TRUE;
	          #errorID := #ALARM_FORCE_PROFILE;
	          #statFBState := #STATE_ERROR;
	        END_IF;
	      ELSE
	        #axis.StatusForceProfile.ActualProfile := 0;
	      END_IF;
	      IF #statFBState <> #STATE_ERROR THEN
	        //call function for force control        
	        #statCommandID := "LSimaHydTO_GetCommandID"(#axis);
	        #axis.Internal.Control.ForceCommand.commandID := #statCommandID;
	        #axis.Internal.Control.ForceCommand.compareMode := #compareMode;
	        #axis.Internal.Control.ForceCommand.conditionMode := #conditionMode;
	        #axis.Internal.Control.ForceCommand.conditionValue := #conditionValue;
	        #axis.Internal.Control.ForceCommand.forceRamp := #forceDerivedValue;
	        #axis.Internal.Control.ForceCommand.forceProfileMode := #forceProfileMode;
	        #axis.Internal.Control.ForceCommand.forceValue := #forceValue;
	        #axis.Internal.Control.ForceCommand.mode := #mode;
	        #axis.Internal.Control.ForceCommand.velocityLimitingValue := #velocityLimitingValue;
	        #axis.Internal.Control.ExecuteForceControl := TRUE;
	        #busy := TRUE;
	        #statFBState := #STATE_BUSY;
	      END_IF;
	    END_IF;
	    
	    
	  #STATE_BUSY:
	    
	    //==================================================================
	    //The command is identified by the commandId.
	    //The FB remains in this state as long as the pos functionality is
	    //active.
	    //==================================================================
	    
	    #statCmdState := "LSimaHydTO_GetAxisForceCommandState"(commandID := #statCommandID, axis := #axis);
	    IF #statCmdState = #MOTION_STATE_EXECUTED THEN
	      #busy := FALSE;
	      #done := TRUE;
	      #statFBState := #STATE_DONE;
	    ELSIF #statCmdState <> #MOTION_STATE_BUFFERED_OR_MOTION OR
	      NOT #axis.StatusActor.Enabled OR #axis.ErrorWord <> 0
	    THEN
	      #busy := FALSE;
	      #commandAborted := TRUE;
	      #statFBState := #STATE_COMMAND_ABORTED;
	    END_IF;
	    
	    
	  #STATE_IDLE:
	    
	    //==================================================================
	    //state analysis (no function)
	    //==================================================================
	    
	    ;
	    
	    
	  #STATE_DONE:
	    
	    //==================================================================
	    //output for one cycle minimum
	    //==================================================================
	    
	    IF NOT #execute  THEN
	      #statFBState := #STATE_IDLE;
	      #done := FALSE;
	    END_IF;
	    
	    
	  #STATE_COMMAND_ABORTED:
	    
	    //==================================================================
	    //reset commandAborted, output for one cycle minimum
	    //==================================================================
	    
	    IF NOT #execute THEN
	      #commandAborted := FALSE;
	      #statFBState := #STATE_IDLE;
	    END_IF;
	    
	    
	  #STATE_ERROR:
	    
	    //==================================================================
	    //reset error, output for one cycle minimum
	    //==================================================================
	
	    IF NOT #execute THEN
	      #error := FALSE;
	      #errorID := #NO_ERROR;
	      #statFBState := #STATE_IDLE;
	    END_IF;
	    
	  ELSE
	    
	    //==================================================================
	    //when FB is busy...
	    //==================================================================
	    
	    ;
	    
	END_CASE;
	
	
	//----------------------------------------------------------------------
	//always executed
	//----------------------------------------------------------------------
	
	#inForceControl := #axis.StatusForce.ForceControl;
	//edge detection
	#statExecuteOld := #execute;
	//------------------------------------------------------------------------------
	
	
END_FUNCTION_BLOCK

FUNCTION_BLOCK "LSimaHydTO_MC_ForceLimiting"
{ S7_Optimized_Access := 'TRUE' }
AUTHOR : APC_ERLF
FAMILY : LSimaHydTO
VERSION : 1.0
   VAR_INPUT 
      execute : Bool;
      forceLimitingProfile : UInt;
      mode : DInt;
      forceProfileMode : DInt;
      conditionMode : DInt := 1;
      compareMode : DInt := 1;
      conditionValue : LReal;
      forceValue : LReal;
      forceDerivedValue : LReal;
      clampingMonitoring : Bool;
      followingErrorDeviation : LReal;
   END_VAR

   VAR_OUTPUT 
      done { ExternalWritable := 'False'} : Bool;
      forceLimited { ExternalWritable := 'False'} : Bool;
      InLimitation { ExternalWritable := 'False'} : Bool;
      inClamping { ExternalWritable := 'False'} : Bool;
      busy { ExternalWritable := 'False'} : Bool;
      commandAborted { ExternalWritable := 'False'} : Bool;
      error { ExternalWritable := 'False'} : Bool;
      errorID { ExternalWritable := 'False'} : Word;
   END_VAR

   VAR_IN_OUT 
      Axis : "LSimaHydTO_typeAxisData";
   END_VAR

   VAR 
      statFBState { ExternalAccessible := 'False'; ExternalVisible := 'False'; ExternalWritable := 'False'} : DInt;
      statCommandID { ExternalAccessible := 'False'; ExternalVisible := 'False'; ExternalWritable := 'False'} : UDInt;
      statCmdState { ExternalAccessible := 'False'; ExternalVisible := 'False'; ExternalWritable := 'False'} : Word;
      statExecuteOld { ExternalAccessible := 'False'; ExternalVisible := 'False'; ExternalWritable := 'False'} : Bool;
   END_VAR

   VAR CONSTANT 
      NO_ERROR : Word := 16#0000;
      STATE_IDLE : DInt;
      STATE_FIRST_CYCLE : DInt := 10;
      STATE_BUSY : DInt := 20;
      STATE_DONE : DInt := 30;
      STATE_COMMAND_ABORTED : DInt := 40;
      STATE_ERROR : DInt := 100;
      MOTION_STATE_NOT_EXISTEND : Word := 16#0000;
      MOTION_STATE_BUFFERED_OR_MOTION : Word := 16#0001;
      MOTION_STATE_EXECUTED : Word := 16#0010;
      MOTION_STATE_ABORTED : Word := 16#0020;
      MOTION_STATE_ERROR : Word := 16#8000;
      NO_ERROR_REACTION : DInt := 0;
      ALARM_AXIS_ERROR_OCCURED : Word := 16#8001;
      ALARM_WRONG_MODE : Word := 16#800A;
      ALARM_AXIS_DISABLED : Word := 16#800F;
      ALARM_FORCE_PROFILE_MODE : Word := 16#80B1;
      ALARM_CONDITION_MODE : Word := 16#80B2;
      ALARM_FORCE_PROFILE : Word := 16#80B3;
      ALARM_COMPARE_MODE : Word := 16#80B4;
      ALARM_FORCE_DERIVED_VALUE : Word := 16#80B5;
   END_VAR


BEGIN
	//================================================================================
	//SIEMENS AG // (c)Copyright 2019 All Rights Reserved
	//--------------------------------------------------------------------------------
	//Library: LSimaHydTO
	//Tested with: S7-15xx
	//Engineering: TIA Portal V15
	//Restrictions: -
	//Requirements: S7-1500 (SW 2.5)
	//Functionality: function to activate/deactivate the force/pressure
	//               limiting of your axis.
	//
	//--------------------------------------------------------------------------------
	//Change log table:
	//
	//Version     Date          Expert in charge    Changes applied
	//01.00.00    15.03.2018    APC_ERLF            First released version
	//================================================================================
	
	
	// ----------------------------------------------------------------------
	// start
	// ----------------------------------------------------------------------
	// rising edge of execute starts functionality
	IF #execute AND NOT #statExecuteOld THEN
	  // initialization
	  #done := FALSE;
	  #commandAborted := FALSE;
	  #forceLimited := FALSE;
	  #busy := FALSE;
	  #error := FALSE;
	  #errorID := #NO_ERROR;
	  #statFBState := #STATE_FIRST_CYCLE;
	END_IF;
	
	// ----------------------------------------------------------------------
	// busy
	// ----------------------------------------------------------------------
	// ------------------------------------------------------------------
	// user implementation begins here
	// example of a state machine
	// ------------------------------------------------------------------
	CASE #statFBState OF
	  #STATE_FIRST_CYCLE:
	    // ==================================================================
	    // This state runs just one time after a rising edge on execute and
	    // calls the function to start the motion.
	    // Get a commandId and buffer it for tracking the command in the
	    // following state STATE_BUSY
	    // ==================================================================
	    // 
	    
	    #commandAborted := FALSE;
	    IF #mode < 0 OR #mode > 2 THEN
	      #error := TRUE;
	      #errorID := #ALARM_WRONG_MODE;
	      #statFBState := #STATE_ERROR;
	    ELSIF #mode <> 0 AND (#forceProfileMode < 0 OR #forceProfileMode > 2) THEN
	      #error := TRUE;
	      #errorID := #ALARM_FORCE_PROFILE_MODE;
	      #statFBState := #STATE_ERROR;
	    ELSIF #mode = 2 AND (#conditionMode < 1 OR #conditionMode > 3) THEN
	      #error := TRUE;
	      #errorID := #ALARM_CONDITION_MODE;
	      #statFBState := #STATE_ERROR;
	    ELSIF #mode = 2 AND #conditionMode > 1 AND (#compareMode < 1 OR #compareMode > 2) THEN
	      #error := TRUE;
	      #errorID := #ALARM_COMPARE_MODE;
	      #statFBState := #STATE_ERROR;
	    ELSIF #mode > 0 AND #forceProfileMode = 0 AND #forceDerivedValue <= 0.0 THEN
	      #error := TRUE;
	      #errorID := #ALARM_FORCE_DERIVED_VALUE;
	      #statFBState := #STATE_ERROR;
	    ELSIF NOT #Axis.StatusActor.Enabled THEN
	      #error := TRUE;
	      #errorID := #ALARM_AXIS_DISABLED;
	      #statFBState := #STATE_ERROR;
	    ELSIF #Axis.#ErrorWord <> 0 AND #Axis.ErrorDetail.Reaction <> #NO_ERROR_REACTION THEN
	      #error := TRUE;
	      #errorID := #ALARM_AXIS_ERROR_OCCURED;
	      #statFBState := #STATE_ERROR;
	    ELSE
	      
	      IF #mode <> 0 AND #forceProfileMode > 0 THEN
	        // check force profile DB 
	        IF #forceLimitingProfile > 0 THEN
	          #Axis.StatusForceProfile.ActualProfile := #forceLimitingProfile;
	        ELSE
	          #Axis.StatusForceProfile.ActualProfile := 0;
	          #error := TRUE;
	          #errorID := #ALARM_FORCE_PROFILE;
	          #statFBState := #STATE_ERROR;
	          
	        END_IF;
	      ELSE
	        #Axis.StatusForceProfile.ActualProfile := 0;
	      END_IF;
	      
	      IF #statFBState <> #STATE_ERROR THEN
	        
	        // call function for force limiting        
	        #statCommandID := "LSimaHydTO_GetCommandID"(#Axis);
	        #Axis.Internal.Control.ForceCommand.commandID := #statCommandID;
	        #Axis.Internal.Control.ForceCommand.compareMode := #compareMode;
	        #Axis.Internal.Control.ForceCommand.conditionMode := #conditionMode;
	        #Axis.Internal.Control.ForceCommand.conditionValue := #conditionValue;
	        #Axis.Internal.Control.ForceCommand.forceRamp := #forceDerivedValue;
	        #Axis.Internal.Control.ForceCommand.forceProfileMode := #forceProfileMode;
	        #Axis.Internal.Control.ForceCommand.forceValue := #forceValue;
	        #Axis.Internal.Control.ForceCommand.mode := #mode;
	        #Axis.Internal.Control.ForceCommand.velocityLimitingValue := 1.0E+12;
	        
	        #Axis.Internal.Control.ForceCommand.clampingMonitoring := #clampingMonitoring;
	        #Axis.Internal.Control.ForceCommand.followingErrorDeviation := #followingErrorDeviation;
	        
	        #Axis.Internal.Control.ExecuteForceLimiting := TRUE;
	        #busy := TRUE;
	        #statFBState := #STATE_BUSY;
	      END_IF;
	    END_IF;
	    
	    
	  #STATE_BUSY:
	    // =================================================================
	    // The  command is identified by the commandId.
	    // The FB remains in this state as long as the pos functionality is active.
	    // ==================================================================
	    #statCmdState := "LSimaHydTO_GetAxisForceCommandState"(commandID := #statCommandID, axis := #Axis);
	    IF #statCmdState = #MOTION_STATE_EXECUTED THEN
	      #busy := FALSE;
	      #done := TRUE;
	      #statFBState := #STATE_DONE;
	      
	    ELSIF #statCmdState <> #MOTION_STATE_BUFFERED_OR_MOTION OR
	      NOT #Axis.StatusActor.Enabled OR #Axis.#ErrorWord <> 0
	    THEN
	      #commandAborted := TRUE;
	      #busy := FALSE;
	      #statFBState := #STATE_COMMAND_ABORTED;
	      
	    END_IF;
	    
	    // -------------------------------------------------------------------------
	    // state analysis (no function)
	    // -------------------------------------------------------------------------
	  #STATE_IDLE:
	    // ======================================================================
	    ;
	    
	  #STATE_DONE:
	    // ======================================================================
	    // output for one cycle minimum
	    IF NOT #execute THEN
	      #statFBState := #STATE_IDLE;
	      #done := FALSE;
	    END_IF;
	    
	  #STATE_COMMAND_ABORTED:
	    // ======================================================================
	    // reset commandAborted, output for one cycle minimum
	    IF NOT #execute THEN
	      #commandAborted := FALSE;
	      #statFBState := #STATE_IDLE;
	    END_IF;
	    
	  #STATE_ERROR:
	    // ======================================================================
	    // reset error, output for one cycle minimum
	    IF NOT #execute THEN
	      #error := FALSE;
	      #errorID := #NO_ERROR;
	      #statFBState := #STATE_IDLE;
	    END_IF;
	    
	    
	  ELSE
	    // ======================================================================
	    // when FB is busy...
	    ;
	END_CASE;
	
	// -------------------------------------------------------------------------
	// always executed
	// -------------------------------------------------------------------------
	#forceLimited := #Axis.StatusForce.ForceLimitingCommand;
	#InLimitation := #Axis.StatusForce.InLimitation;
	#inClamping := #Axis.StatusForce.InClamping;
	
	// edge detection
	#statExecuteOld := #execute;
	
	// ------------------------------------------------------------------------------
END_FUNCTION_BLOCK

FUNCTION "LSimaHydTO_UnscaleDriveDWord" : DWord
{ S7_Optimized_Access := 'TRUE' }
AUTHOR : APC_ERLF
FAMILY : LSimaHydTO
VERSION : 1.0
   VAR_INPUT 
      reference : LReal;
      value : LReal;
   END_VAR

   VAR_TEMP 
      tempNormValue : LReal;
   END_VAR


BEGIN
	//================================================================================
	//SIEMENS AG // (c)Copyright 2019 All Rights Reserved
	//--------------------------------------------------------------------------------
	//Library:       LSimaHydTO
	//Tested with:   S7-15xx
	//Engineering:   TIA Portal  V15
	//Restrictions:  -
	//Requirements:  S7-1500 (FW 2.5)
	//Functionality: - for internal use
	//
	//--------------------------------------------------------------------------------
	//Change log table:
	//
	//Version     Date          Expert in charge    Changes applied
	//01.00.00    15.03.2018    APC_ERLF            First released version
	//================================================================================
	
	
	#tempNormValue := LIMIT(MN := -2.0, IN := #value / #reference, MX := 1.999999999);
	#LSimaHydTO_UnscaleDriveDWord := DINT_TO_DWORD(LREAL_TO_DINT(#tempNormValue * 1073741824.0));
	
	
END_FUNCTION

FUNCTION "SimaHydTO_ChangeLog" : Void
{ S7_Optimized_Access := 'TRUE' }
AUTHOR : APC_ERLF
FAMILY : SimaHydTO
VERSION : 1.22

BEGIN
	//================================================================================
	//SIEMENS AG // (c)Copyright 2020 All Rights Reserved
	//--------------------------------------------------------------------------------
	//Library: LSimaHydTO
	//Tested with: S7-15xx
	//Engineering: TIA Portal  V15
	//Restrictions: -
	//Requirements: S7-1500 (SW 2.5)
	//Functionality: none, change log only   
	//
	//--------------------------------------------------------------------------------
	//Change log table:
	//
	//Version     Date          Expert in charge    Changes applied
	//01.19    23.01.2020    APC_ERLF            First released version
	//
	//01.20    30.01.2020    APC_ERLF           LSimaHydTO_HydAxis: - fixed: homing causes puls on QOutput
	//
	//01.21    11.03.2020    APC_ERLF           HMI functions: - fixed:Vchar assignment is not saved in parameter editor after "Activate". 
	//
	//01.22    28.04.2020    APC_ERLF           LSimaHydTO_HydAxis; LSimaHydTO_MC_MoveAbsOpenLoop, 
	//                                          LSimaHydTO_GetCharacteristic, Simulation     - improved: units are taken into account for the control
	//
	//===============================================================================
	
END_FUNCTION

DATA_BLOCK "HydAxisAnalog1VChar"   // DB33140
{ S7_Optimized_Access := 'TRUE' }
FAMILY : SimaHydTO
VERSION : 1.0
// stored: AutoNumber true, DBAccessibleFromOPCUA true, InstanceOfName LSimaHydTO_typeVCharData, InstanceOfType UDT, IsOnlyStoredInLoadMemory false, IsWriteProtectedInAS false
"LSimaHydTO_typeVCharData"
BEGIN
   QOutput[0] := -100.0;
   QOutput[1] := 0.0;
   QOutput[2] := 100.0;
   Velocity[0] := -100.0;
   Velocity[1] := 0.0;
   Velocity[2] := 100.0;
END_DATA_BLOCK

DATA_BLOCK "HydAxisAnalog1_Data"   // DB33130
{ S7_Optimized_Access := 'TRUE' }
FAMILY : SimaHydTO
VERSION : 1.0
// stored: AutoNumber true, DBAccessibleFromOPCUA true, InstanceOfName LSimaHydTO_typeAxisData, InstanceOfType UDT, IsOnlyStoredInLoadMemory false, IsWriteProtectedInAS false
"LSimaHydTO_typeAxisData"
BEGIN
   Actor.DirectionValves.DelayTimeValveForward := 0.01;
   Actor.DirectionValves.DelayTimeValveBackward := 0.01;
   Actor.DirectionValves.ValvesOffMode := 1;
   ValveCharacteristic.DB_NUMBER := 33140;
END_DATA_BLOCK

DATA_BLOCK "HydAxisAnalog2VChar"   // DB33141
{ S7_Optimized_Access := 'TRUE' }
FAMILY : SimaHydTO
VERSION : 1.0
// stored: AutoNumber true, DBAccessibleFromOPCUA true, InstanceOfName LSimaHydTO_typeVCharData, InstanceOfType UDT, IsOnlyStoredInLoadMemory false, IsWriteProtectedInAS false
"LSimaHydTO_typeVCharData"
BEGIN
   QOutput[0] := -100.0;
   QOutput[1] := 0.0;
   QOutput[2] := 100.0;
   Velocity[0] := -100.0;
   Velocity[1] := 0.0;
   Velocity[2] := 100.0;
END_DATA_BLOCK

DATA_BLOCK "HydAxisAnalog2_Data"   // DB33131
{ S7_Optimized_Access := 'TRUE' }
FAMILY : SimaHydTO
VERSION : 1.0
// stored: AutoNumber true, DBAccessibleFromOPCUA true, InstanceOfName LSimaHydTO_typeAxisData, InstanceOfType UDT, IsOnlyStoredInLoadMemory false, IsWriteProtectedInAS false
"LSimaHydTO_typeAxisData"
BEGIN
   ValveCharacteristic.DB_NUMBER := 33141;
END_DATA_BLOCK

DATA_BLOCK "HydAxisDriveSimulationVChar"   // DB33172
{ S7_Optimized_Access := 'TRUE' }
FAMILY : SimaHydTO
VERSION : 1.0
// stored: AutoNumber true, DBAccessibleFromOPCUA true, InstanceOfName LSimaHydTO_typeVCharData, InstanceOfType UDT, IsOnlyStoredInLoadMemory false, IsWriteProtectedInAS false
"LSimaHydTO_typeVCharData"
BEGIN
   QOutput[0] := -200.0;
   QOutput[1] := 0.0;
   QOutput[2] := 200.0;
   Velocity[0] := -200.0;
   Velocity[1] := 0.0;
   Velocity[2] := 200.0;
END_DATA_BLOCK

DATA_BLOCK "HydAxisDriveVChar"   // DB33142
{ S7_Optimized_Access := 'TRUE' }
FAMILY : SimaHydTO
VERSION : 1.0
// stored: AutoNumber true, DBAccessibleFromOPCUA true, InstanceOfName LSimaHydTO_typeVCharData, InstanceOfType UDT, IsOnlyStoredInLoadMemory false, IsWriteProtectedInAS false
"LSimaHydTO_typeVCharData"
BEGIN
   QOutput[0] := -100.0;
   QOutput[1] := 0.0;
   QOutput[2] := 100.0;
   Velocity[0] := -100.0;
   Velocity[1] := 0.0;
   Velocity[2] := 100.0;
END_DATA_BLOCK

DATA_BLOCK "HydAxisDrive_Data"   // DB33132
{ S7_Optimized_Access := 'TRUE' }
FAMILY : SimaHydTO
VERSION : 1.0
// stored: AutoNumber true, DBAccessibleFromOPCUA true, InstanceOfName LSimaHydTO_typeAxisData, InstanceOfType UDT, IsOnlyStoredInLoadMemory false, IsWriteProtectedInAS false
"LSimaHydTO_typeAxisData"
BEGIN
   ValveCharacteristic.DB_NUMBER := 33142;
   ValveCharacteristic.SmoothChangeTime := 0.04;
   Pressure_A_Transducer.Area := 1256.63696;
   Pressure_B_Transducer.Area := 640.884992275975;
   SmoothingFilter.VelocityFilter := 0.02;
END_DATA_BLOCK

DATA_BLOCK "HydAxisSimulationVChar1"   // DB33170
{ S7_Optimized_Access := 'TRUE' }
FAMILY : SimaHydTO
VERSION : 1.0
// stored: AutoNumber true, DBAccessibleFromOPCUA true, InstanceOfName LSimaHydTO_typeVCharData, InstanceOfType UDT, IsOnlyStoredInLoadMemory false, IsWriteProtectedInAS false
"LSimaHydTO_typeVCharData"
BEGIN
   QOutput[0] := -100.0;
   QOutput[1] := -30.0;
   QOutput[2] := 0.0;
   QOutput[3] := 30.0;
   QOutput[4] := 100.0;
   Velocity[0] := -100.0;
   Velocity[1] := -50.0;
   Velocity[2] := 0.0;
   Velocity[3] := 40.0;
   Velocity[4] := 100.0;
END_DATA_BLOCK

DATA_BLOCK "HydAxisSimulationVChar2"   // DB33171
{ S7_Optimized_Access := 'TRUE' }
FAMILY : SimaHydTO
VERSION : 1.0
// stored: AutoNumber true, DBAccessibleFromOPCUA true, InstanceOfName LSimaHydTO_typeVCharData, InstanceOfType UDT, IsOnlyStoredInLoadMemory false, IsWriteProtectedInAS false
"LSimaHydTO_typeVCharData"
BEGIN
   QOutput[0] := -100.0;
   QOutput[1] := -30.0;
   QOutput[2] := 0.0;
   QOutput[3] := 30.0;
   QOutput[4] := 100.0;
   Velocity[0] := -100.0;
   Velocity[1..3] := 0.0;
   Velocity[4] := 100.0;
END_DATA_BLOCK

DATA_BLOCK "InstHydAxisCallFB_Analog1"   // DB33120
{ DB_Accessible_From_OPC_UA := 'FALSE' }
FAMILY : SimaHydTO
VERSION : 1.0
// stored: AutoNumber true, DBAccessibleFromOPCUA false, InstanceOfName LSimaHydTO_HydAxisCall, InstanceOfType FB
"LSimaHydTO_HydAxisCall"
BEGIN
END_DATA_BLOCK

DATA_BLOCK "InstHydAxisCallFB_Analog2"   // DB33121
{ DB_Accessible_From_OPC_UA := 'FALSE' }
FAMILY : SimaHydTO
VERSION : 1.0
// stored: AutoNumber true, DBAccessibleFromOPCUA false, InstanceOfName LSimaHydTO_HydAxisCall, InstanceOfType FB
"LSimaHydTO_HydAxisCall"
BEGIN
END_DATA_BLOCK

DATA_BLOCK "InstHydAxisCallFB_Drive"   // DB33122
{ DB_Accessible_From_OPC_UA := 'FALSE' }
FAMILY : SimaHydTO
VERSION : 1.0
// stored: AutoNumber true, DBAccessibleFromOPCUA false, InstanceOfName LSimaHydTO_HydAxisCall, InstanceOfType FB
"LSimaHydTO_HydAxisCall"
BEGIN
END_DATA_BLOCK

DATA_BLOCK "InstHydraulicsSimulationAnalog1"   // DB33160
{ DB_Accessible_From_OPC_UA := 'FALSE' }
FAMILY : SimaHydTO
VERSION : 1.0
// stored: AutoNumber true, DBAccessibleFromOPCUA false, InstanceOfName LSimaHydTO_HydraulicSimulationAnalog, InstanceOfType FB
"LSimaHydTO_HydraulicSimulationAnalog"
BEGIN
END_DATA_BLOCK

DATA_BLOCK "InstHydraulicsSimulationAnalog2"   // DB33161
{ DB_Accessible_From_OPC_UA := 'FALSE' }
FAMILY : SimaHydTO
VERSION : 1.0
// stored: AutoNumber true, DBAccessibleFromOPCUA false, InstanceOfName LSimaHydTO_HydraulicSimulationAnalog, InstanceOfType FB
"LSimaHydTO_HydraulicSimulationAnalog"
BEGIN
END_DATA_BLOCK

DATA_BLOCK "InstHydraulicsSimulationDrive"   // DB33162
{ DB_Accessible_From_OPC_UA := 'FALSE' }
FAMILY : SimaHydTO
VERSION : 1.0
// stored: AutoNumber true, DBAccessibleFromOPCUA false, InstanceOfName LSimaHydTO_HydraulicSimulationDrive, InstanceOfType FB
"LSimaHydTO_HydraulicSimulationDrive"
BEGIN
END_DATA_BLOCK

DATA_BLOCK "InstSimaHydTO_HMI"   // DB33105
TITLE = InstSimaHydTO_HMI
{ DB_Accessible_From_OPC_UA := 'FALSE' }
FAMILY : SimaHydTO
VERSION : 1.0
// Instance data block
// stored: AutoNumber true, DBAccessibleFromOPCUA false, InstanceOfName SimaHydTO_HMI, InstanceOfType FB
"SimaHydTO_HMI"
BEGIN
END_DATA_BLOCK

DATA_BLOCK "LSimaHydTO_MC_ForceControl_DB"   // DB1
AUTHOR : APC_ERLF
FAMILY : LSimaHydTO
VERSION : 1.0
// stored: AutoNumber true, DBAccessibleFromOPCUA true, InstanceOfName LSimaHydTO_MC_ForceControl, InstanceOfType FB
"LSimaHydTO_MC_ForceControl"
BEGIN
END_DATA_BLOCK

DATA_BLOCK "MasterCharacteristics_01"   // DB6001
{ S7_Optimized_Access := 'TRUE' }
FAMILY : SimaHydTO
VERSION : 1.0
// stored: AutoNumber true, DBAccessibleFromOPCUA true, InstanceOfName LSimaHydTO_typeVCharData, InstanceOfType UDT, IsOnlyStoredInLoadMemory false, IsWriteProtectedInAS false
"LSimaHydTO_typeVCharData"
BEGIN
   QOutput[0] := -100.0;
   QOutput[1] := -50.0;
   QOutput[2] := 0.0;
   QOutput[3] := 50.0;
   QOutput[4] := 100.0;
   Velocity[0] := -100.0;
   Velocity[1] := -30.0;
   Velocity[2] := 0.0;
   Velocity[3] := 40.0;
   Velocity[4] := 100.0;
END_DATA_BLOCK

DATA_BLOCK "SimaHydTO_AdvancedAxisControl_DB"   // DB4
FAMILY : SimaHydTO
VERSION : 1.0
// stored: AutoNumber true, DBAccessibleFromOPCUA true, InstanceOfName SimaHydTO_AdvancedAxisControl, InstanceOfType FB
"SimaHydTO_AdvancedAxisControl"
BEGIN
END_DATA_BLOCK

DATA_BLOCK "SimaHydTO_AdvancedAxisControl_DB_1"   // DB8
FAMILY : SimaHydTO
VERSION : 1.0
// stored: AutoNumber true, DBAccessibleFromOPCUA true, InstanceOfName SimaHydTO_AdvancedAxisControl, InstanceOfType FB
"SimaHydTO_AdvancedAxisControl"
BEGIN
END_DATA_BLOCK

DATA_BLOCK "SimaHydTO_AxisAdvanced_PosAxis_DB"   // DB5
FAMILY : SimaHydTO/LAxisBasics
VERSION : 1.0
// stored: AutoNumber true, DBAccessibleFromOPCUA true, InstanceOfName SimaHydTO_AxisAdvanced_PosAxis, InstanceOfType FB
"SimaHydTO_AxisAdvanced_PosAxis"
BEGIN
END_DATA_BLOCK

DATA_BLOCK "SimaHydTO_AxisAdvanced_PosAxis_DB_1"   // DB9
FAMILY : SimaHydTO/LAxisBasics
VERSION : 1.0
// stored: AutoNumber true, DBAccessibleFromOPCUA true, InstanceOfName SimaHydTO_AxisAdvanced_PosAxis, InstanceOfType FB
"SimaHydTO_AxisAdvanced_PosAxis"
BEGIN
END_DATA_BLOCK

DATA_BLOCK "SimaHydTO_AxisAdvanced_SyncAxis_DB"   // DB6
FAMILY : SimaHydTO/LAxisBasics
VERSION : 1.0
// stored: AutoNumber true, DBAccessibleFromOPCUA true, InstanceOfName SimaHydTO_AxisAdvanced_SyncAxis, InstanceOfType FB
"SimaHydTO_AxisAdvanced_SyncAxis"
BEGIN
END_DATA_BLOCK

DATA_BLOCK "SimaHydTO_AxisBasics_PosAxis_DB"   // DB2
FAMILY : SimaHydTO/LAxisBasics
VERSION : 1.0
// stored: AutoNumber true, DBAccessibleFromOPCUA true, InstanceOfName SimaHydTO_AxisBasics_PosAxis, InstanceOfType FB
"SimaHydTO_AxisBasics_PosAxis"
BEGIN
END_DATA_BLOCK

DATA_BLOCK "SimaHydTO_HMIConnection"   // DB33100
TITLE = SimaHydTO_HMIConnection
{ S7_Optimized_Access := 'TRUE' }
FAMILY : SimaHydTO
VERSION : 1.0
// Connection data to HMI
// stored: AutoNumber true, DBAccessibleFromOPCUA true, InstanceOfName SimaHydTO_typeHMIConnection, InstanceOfType UDT, IsOnlyStoredInLoadMemory false, IsWriteProtectedInAS false
"SimaHydTO_typeHMIConnection"
BEGIN
   GetCharacteristics.ConfigData.safetyDistance := 100.0;
END_DATA_BLOCK

DATA_BLOCK "TestCharacteristics_01"   // DB5001
{ S7_Optimized_Access := 'TRUE' }
FAMILY : SimaHydTO
VERSION : 1.0
// stored: AutoNumber true, DBAccessibleFromOPCUA true, InstanceOfName LSimaHydTO_typeVCharData, InstanceOfType UDT, IsOnlyStoredInLoadMemory false, IsWriteProtectedInAS false
"LSimaHydTO_typeVCharData"
BEGIN
END_DATA_BLOCK

DATA_BLOCK "TestCharacteristics_02"   // DB5002
{ S7_Optimized_Access := 'TRUE' }
FAMILY : SimaHydTO
VERSION : 1.0
// stored: AutoNumber true, DBAccessibleFromOPCUA true, InstanceOfName LSimaHydTO_typeVCharData, InstanceOfType UDT, IsOnlyStoredInLoadMemory false, IsWriteProtectedInAS false
"LSimaHydTO_typeVCharData"
BEGIN
END_DATA_BLOCK

DATA_BLOCK "TestCharacteristics_03"   // DB5003
{ S7_Optimized_Access := 'TRUE' }
FAMILY : SimaHydTO
VERSION : 1.0
// stored: AutoNumber true, DBAccessibleFromOPCUA true, InstanceOfName LSimaHydTO_typeVCharData, InstanceOfType UDT, IsOnlyStoredInLoadMemory false, IsWriteProtectedInAS false
"LSimaHydTO_typeVCharData"
BEGIN
END_DATA_BLOCK

DATA_BLOCK "TestCharacteristics_04"   // DB5004
{ S7_Optimized_Access := 'TRUE' }
FAMILY : SimaHydTO
VERSION : 1.0
// stored: AutoNumber true, DBAccessibleFromOPCUA true, InstanceOfName LSimaHydTO_typeVCharData, InstanceOfType UDT, IsOnlyStoredInLoadMemory false, IsWriteProtectedInAS false
"LSimaHydTO_typeVCharData"
BEGIN
END_DATA_BLOCK

DATA_BLOCK "TestCharacteristics_05"   // DB5005
{ S7_Optimized_Access := 'TRUE' }
FAMILY : SimaHydTO
VERSION : 1.0
// stored: AutoNumber true, DBAccessibleFromOPCUA true, InstanceOfName LSimaHydTO_typeVCharData, InstanceOfType UDT, IsOnlyStoredInLoadMemory false, IsWriteProtectedInAS false
"LSimaHydTO_typeVCharData"
BEGIN
END_DATA_BLOCK

DATA_BLOCK "TestCharacteristics_06"   // DB5006
{ S7_Optimized_Access := 'TRUE' }
FAMILY : SimaHydTO
VERSION : 1.0
// stored: AutoNumber true, DBAccessibleFromOPCUA true, InstanceOfName LSimaHydTO_typeVCharData, InstanceOfType UDT, IsOnlyStoredInLoadMemory false, IsWriteProtectedInAS false
"LSimaHydTO_typeVCharData"
BEGIN
END_DATA_BLOCK

DATA_BLOCK "IEC_Timer_0_DB"   // DB7
{ S7_Optimized_Access := 'TRUE' }
// stored: AutoNumber true, DBAccessibleFromOPCUA true, InstanceOfName IEC_TIMER, OfSystemLibElement IEC_TIMER, OfSystemLibVersion 1.0
"IEC_TIMER"
   // VAR
   //    PT : Time;
   //    ET { ExternalWritable := 'False'} : Time;
   //    IN : Bool;
   //    Q { ExternalWritable := 'False'} : Bool;
   // END_VAR
BEGIN
END_DATA_BLOCK

DATA_BLOCK "IEC_Timer_0_DB_1"   // DB10
{ S7_Optimized_Access := 'TRUE' }
// stored: AutoNumber true, DBAccessibleFromOPCUA true, InstanceOfName IEC_TIMER, OfSystemLibElement IEC_TIMER, OfSystemLibVersion 1.0
"IEC_TIMER"
   // VAR
   //    PT : Time;
   //    ET { ExternalWritable := 'False'} : Time;
   //    IN : Bool;
   //    Q { ExternalWritable := 'False'} : Bool;
   // END_VAR
BEGIN
END_DATA_BLOCK

DATA_BLOCK "IEC_Timer_0_DB_2"   // DB11
{ S7_Optimized_Access := 'TRUE' }
// stored: AutoNumber true, DBAccessibleFromOPCUA true, InstanceOfName IEC_TIMER, OfSystemLibElement IEC_TIMER, OfSystemLibVersion 1.0
"IEC_TIMER"
   // VAR
   //    PT : Time;
   //    ET { ExternalWritable := 'False'} : Time;
   //    IN : Bool;
   //    Q { ExternalWritable := 'False'} : Bool;
   // END_VAR
BEGIN
END_DATA_BLOCK

DATA_BLOCK "IEC_Timer_0_DB_3"   // DB12
{ S7_Optimized_Access := 'TRUE' }
// stored: AutoNumber true, DBAccessibleFromOPCUA true, InstanceOfName IEC_TIMER, OfSystemLibElement IEC_TIMER, OfSystemLibVersion 1.0
"IEC_TIMER"
   // VAR
   //    PT : Time;
   //    ET { ExternalWritable := 'False'} : Time;
   //    IN : Bool;
   //    Q { ExternalWritable := 'False'} : Bool;
   // END_VAR
BEGIN
END_DATA_BLOCK
